LIN {X 0,Y 249.052,Z 167.452,A -85,B 0,C 180,E1 -18878.627,E2 -18878.627} C_VEL
LIN {X 0,Y 249.159,Z 167.445,A -85,B 0,C 180,E1 -18883.615,E2 -18883.615} C_VEL
LIN {X 0,Y 249.22,Z 167.437,A -85,B 0,C 180,E1 -18888.614,E2 -18888.614} C_VEL
LIN {X 0,Y 249.416,Z 167.401,A -85,B 0,C 180,E1 -18891.9,E2 -18891.9} C_VEL
LIN {X 0,Y 249.265,Z 167.429,A -85,B 0,C 180,E1 -18895.147,E2 -18895.147} C_VEL
LIN {X 0,Y 249.662,Z 167.381,A -85,B 0,C 180,E1 -18898.386,E2 -18898.386} C_VEL
LIN {X 0,Y 249.67,Z 167.37,A -85,B 0,C 180,E1 -18901.612,E2 -18901.612} C_VEL
LIN {X 0,Y 249.428,Z 167.402,A -85,B 0,C 180,E1 -18906.546,E2 -18906.546} C_VEL
LIN {X 0,Y 249.344,Z 167.415,A -85,B 0,C 180,E1 -18909.736,E2 -18909.736} C_VEL
LIN {X 0,Y 249.183,Z 167.435,A -85,B 0,C 180,E1 -18914.704,E2 -18914.704} C_VEL
LIN {X 0,Y 249.118,Z 167.445,A -85,B 0,C 180,E1 -18918.078,E2 -18918.078} C_VEL
LIN {X 0,Y 249.083,Z 167.452,A -85,B 0,C 180,E1 -18921.518,E2 -18921.518} C_VEL
LIN {X 0,Y 249.117,Z 167.45,A -85,B 0,C 180,E1 -18925.475,E2 -18925.475} C_VEL
LIN {X 0,Y 249.05,Z 167.46,A -85,B 0,C 180,E1 -18930.102,E2 -18930.102} C_VEL
LIN {X 0,Y 249.071,Z 167.695,A -85,B 0,C 180,E1 -18930.523,E2 -18930.523} C_VEL
LIN {X 0,Y 249.432,Z 169.077,A -85,B 0,C 180,E1 -18931.179,E2 -18931.179} C_VEL
LIN {X 0,Y 252.028,Z 173,A -85,B 0,C 180,E1 -18931.947,E2 -18931.947} C_VEL
LIN {X 0,Y 253.509,Z 175.144,A -85,B 0,C 180,E1 -18932.37,E2 -18932.37} C_VEL
LIN {X 0,Y 260.713,Z 186.536,A -85,B 0,C 180,E1 -18934.354,E2 -18934.354} C_VEL
LIN {X 0,Y 269.126,Z 201.959,A -85,B 0,C 180,E1 -18936.505,E2 -18936.505} C_VEL
LIN {X 0,Y 275.328,Z 215.39,A -85,B 0,C 180,E1 -18938.036,E2 -18938.036} C_VEL
LIN {X 0,Y 272.536,Z 275.676,A -85,B 0,C 180,E1 -18939.662,E2 -18939.662} C_VEL
LIN {X 0,Y 271.152,Z 289.633,A -85,B 0,C 180,E1 -18940.333,E2 -18940.333} C_VEL
LIN {X 0,Y 269.51,Z 302.431,A -85,B 0,C 180,E1 -18941.293,E2 -18941.293} C_VEL
LIN {X 0,Y 267.486,Z 313.271,A -85,B 0,C 180,E1 -18942.357,E2 -18942.357} C_VEL
LIN {X 0,Y 265.177,Z 324.055,A -85,B 0,C 180,E1 -18943.733,E2 -18943.733} C_VEL
LIN {X 0,Y 262.562,Z 334.24,A -85,B 0,C 180,E1 -18945.361,E2 -18945.361} C_VEL
LIN {X 0,Y 259.944,Z 343.294,A -85,B 0,C 180,E1 -18947.168,E2 -18947.168} C_VEL
LIN {X 0,Y 257.103,Z 352.123,A -85,B 0,C 180,E1 -18949.396,E2 -18949.396} C_VEL
LIN {X 0,Y 254.695,Z 359.121,A -85,B 0,C 180,E1 -18951.621,E2 -18951.621} C_VEL
LIN {X 0,Y 252.375,Z 365.518,A -85,B 0,C 180,E1 -18954.211,E2 -18954.211} C_VEL
LIN {X 0,Y 250.551,Z 370.339,A -85,B 0,C 180,E1 -18956.782,E2 -18956.782} C_VEL
LIN {X 0,Y 249.074,Z 374.017,A -85,B 0,C 180,E1 -18959.476,E2 -18959.476} C_VEL
LIN {X 0,Y 248.275,Z 375.843,A -85,B 0,C 180,E1 -18961.344,E2 -18961.344} C_VEL
LIN {X 0,Y 247.697,Z 377.032,A -85,B 0,C 180,E1 -18963.001,E2 -18963.001} C_VEL
LIN {X 0,Y 247.134,Z 377.998,A -85,B 0,C 180,E1 -18965.505,E2 -18965.505} C_VEL
LIN {X 0,Y 246.776,Z 378.012,A -85,B 0,C 180,E1 -18968.27,E2 -18968.27} C_VEL
LIN {X 0,Y 246.746,Z 377.407,A -85,B 0,C 180,E1 -18970.037,E2 -18970.037} C_VEL
LIN {X 0,Y 246.719,Z 376.398,A -85,B 0,C 180,E1 -18971.739,E2 -18971.739} C_VEL
LIN {X 0,Y 246.848,Z 374.953,A -85,B 0,C 180,E1 -18973.459,E2 -18973.459} C_VEL
LIN {X 0,Y 247.272,Z 371.847,A -85,B 0,C 180,E1 -18976.048,E2 -18976.048} C_VEL
LIN {X 0,Y 247.792,Z 367.733,A -85,B 0,C 180,E1 -18978.549,E2 -18978.549} C_VEL
LIN {X 0,Y 248.725,Z 361.306,A -85,B 0,C 180,E1 -18981.473,E2 -18981.473} C_VEL
LIN {X 0,Y 249.811,Z 354.327,A -85,B 0,C 180,E1 -18983.944,E2 -18983.944} C_VEL
LIN {X 0,Y 250.983,Z 347.179,A -85,B 0,C 180,E1 -18985.986,E2 -18985.986} C_VEL
LIN {X 0,Y 252.381,Z 338.546,A -85,B 0,C 180,E1 -18988.005,E2 -18988.005} C_VEL
LIN {X 0,Y 254.085,Z 327.819,A -85,B 0,C 180,E1 -18990,E2 -18990} C_VEL
LIN {X 0,Y 255.511,Z 317.218,A -85,B 0,C 180,E1 -18991.576,E2 -18991.576} C_VEL
LIN {X 0,Y 256.936,Z 305.486,A -85,B 0,C 180,E1 -18992.94,E2 -18992.94} C_VEL
LIN {X 0,Y 258.068,Z 293.324,A -85,B 0,C 180,E1 -18994.002,E2 -18994.002} C_VEL
LIN {X 0,Y 258.95,Z 280.161,A -85,B 0,C 180,E1 -18994.817,E2 -18994.817} C_VEL
LIN {X 0,Y 259.553,Z 267.449,A -85,B 0,C 180,E1 -18995.292,E2 -18995.292} C_VEL
LIN {X 0,Y 261.586,Z 201.975,A -85,B 0,C 180,E1 -18997.076,E2 -18997.076} C_VEL
LIN {X 0,Y 259.605,Z 195.135,A -85,B 0,C 180,E1 -18997.457,E2 -18997.457} C_VEL
LIN {X 0,Y 251.738,Z 173.167,A -85,B 0,C 180,E1 -18998.873,E2 -18998.873} C_VEL
LIN {X 0,Y 249.492,Z 168.039,A -85,B 0,C 180,E1 -18999.256,E2 -18999.256} C_VEL
LIN {X 0,Y 249.385,Z 167.421,A -85,B 0,C 180,E1 -18999.296,E2 -18999.296} C_VEL
LIN {X 0,Y 249.138,Z 167.452,A -85,B 0,C 180,E1 -19004.708,E2 -19004.708} C_VEL
LIN {X 0,Y 249.072,Z 167.46,A -85,B 0,C 180,E1 -19008.083,E2 -19008.083} C_VEL
LIN {X 0,Y 249.038,Z 167.46,A -85,B 0,C 180,E1 -19011.523,E2 -19011.523} C_VEL
LIN {X 0,Y 249.035,Z 167.435,A -85,B 0,C 180,E1 -19015.438,E2 -19015.438} C_VEL
LIN {X 0,Y 249.021,Z 167.457,A -85,B 0,C 180,E1 -19018.969,E2 -19018.969} C_VEL
LIN {X 0,Y 249.023,Z 167.464,A -85,B 0,C 180,E1 -19022.428,E2 -19022.428} C_VEL
LIN {X 0,Y 249.024,Z 167.451,A -85,B 0,C 180,E1 -19026.347,E2 -19026.347} C_VEL
LIN {X 0,Y 248.977,Z 167.47,A -85,B 0,C 180,E1 -19030.485,E2 -19030.485} C_VEL
LIN {X 0,Y 248.96,Z 167.462,A -85,B 0,C 180,E1 -19034.89,E2 -19034.89} C_VEL
LIN {X 0,Y 248.978,Z 167.455,A -85,B 0,C 180,E1 -19037.356,E2 -19037.356} C_VEL
LIN {X 0,Y 249.04,Z 167.461,A -85,B 0,C 180,E1 -19042.202,E2 -19042.202} C_VEL
LIN {X 0,Y 249.043,Z 167.457,A -85,B 0,C 180,E1 -19045.64,E2 -19045.64} C_VEL
LIN {X 0,Y 248.994,Z 167.445,A -85,B 0,C 180,E1 -19049.466,E2 -19049.466} C_VEL
LIN {X 0,Y 249.014,Z 167.455,A -85,B 0,C 180,E1 -19053.156,E2 -19053.156} C_VEL
LIN {X 0,Y 249.006,Z 167.467,A -85,B 0,C 180,E1 -19056.726,E2 -19056.726} C_VEL
LIN {X 0,Y 249.042,Z 167.463,A -85,B 0,C 180,E1 -19060.207,E2 -19060.207} C_VEL
LIN {X 0,Y 249.16,Z 167.442,A -85,B 0,C 180,E1 -19063.617,E2 -19063.617} C_VEL
LIN {X 0,Y 249.218,Z 167.439,A -85,B 0,C 180,E1 -19068.616,E2 -19068.616} C_VEL
LIN {X 0,Y 249.418,Z 167.41,A -85,B 0,C 180,E1 -19071.902,E2 -19071.902} C_VEL
LIN {X 0,Y 249.259,Z 167.435,A -85,B 0,C 180,E1 -19075.149,E2 -19075.149} C_VEL
LIN {X 0,Y 249.658,Z 167.381,A -85,B 0,C 180,E1 -19078.388,E2 -19078.388} C_VEL
LIN {X 0,Y 249.66,Z 167.384,A -85,B 0,C 180,E1 -19081.614,E2 -19081.614} C_VEL
LIN {X 0,Y 249.429,Z 167.411,A -85,B 0,C 180,E1 -19086.472,E2 -19086.472} C_VEL
LIN {X 0,Y 249.402,Z 167.412,A -85,B 0,C 180,E1 -19088.405,E2 -19088.405} C_VEL
LIN {X 0,Y 248.673,Z 167.508,A -85,B 0,C 180,E1 -19089.751,E2 -19089.751} C_VEL
LIN {X 0,Y 245.735,Z 167.876,A -85,B 0,C 180,E1 -19091.942,E2 -19091.942} C_VEL
LIN {X 0,Y 243.258,Z 168.185,A -85,B 0,C 180,E1 -19093.726,E2 -19093.726} C_VEL
LIN {X 0,Y 242.186,Z 168.315,A -85,B 0,C 180,E1 -19095.112,E2 -19095.112} C_VEL
LIN {X 0,Y 242.093,Z 168.323,A -85,B 0,C 180,E1 -19095.583,E2 -19095.583} C_VEL
LIN {X 0,Y 241.989,Z 168.34,A -85,B 0,C 180,E1 -19100.397,E2 -19100.397} C_VEL
LIN {X 0,Y 242.028,Z 168.335,A -85,B 0,C 180,E1 -19103.988,E2 -19103.988} C_VEL
LIN {X 0,Y 241.972,Z 168.342,A -85,B 0,C 180,E1 -19107.693,E2 -19107.693} C_VEL
LIN {X 0,Y 241.957,Z 168.345,A -85,B 0,C 180,E1 -19111.524,E2 -19111.524} C_VEL
LIN {X 0,Y 241.982,Z 168.342,A -85,B 0,C 180,E1 -19115.588,E2 -19115.588} C_VEL
LIN {X 0,Y 241.944,Z 168.348,A -85,B 0,C 180,E1 -19119.723,E2 -19119.723} C_VEL
LIN {X 0,Y 241.901,Z 168.355,A -85,B 0,C 180,E1 -19124.21,E2 -19124.21} C_VEL
LIN {X 0,Y 241.922,Z 168.351,A -85,B 0,C 180,E1 -19128.074,E2 -19128.074} C_VEL
LIN {X 0,Y 241.99,Z 168.339,A -85,B 0,C 180,E1 -19132.417,E2 -19132.417} C_VEL
LIN {X 0,Y 242.046,Z 168.546,A -85,B 0,C 180,E1 -19134.754,E2 -19134.754} C_VEL
LIN {X 0,Y 244.315,Z 179.21,A -85,B 0,C 180,E1 -19138.815,E2 -19138.815} C_VEL
LIN {X 0,Y 245.111,Z 183.189,A -85,B 0,C 180,E1 -19140.272,E2 -19140.272} C_VEL
LIN {X 0,Y 249.449,Z 195.846,A -85,B 0,C 180,E1 -19141.11,E2 -19141.11} C_VEL
LIN {X 0,Y 254.127,Z 234.244,A -85,B 0,C 180,E1 -19142.738,E2 -19142.738} C_VEL
LIN {X 0,Y 252.285,Z 292.507,A -85,B 0,C 180,E1 -19144.418,E2 -19144.418} C_VEL
LIN {X 0,Y 251.321,Z 306.261,A -85,B 0,C 180,E1 -19145.144,E2 -19145.144} C_VEL
LIN {X 0,Y 249.948,Z 319.146,A -85,B 0,C 180,E1 -19146.159,E2 -19146.159} C_VEL
LIN {X 0,Y 248.279,Z 331.738,A -85,B 0,C 180,E1 -19147.533,E2 -19147.533} C_VEL
LIN {X 0,Y 246.562,Z 342.976,A -85,B 0,C 180,E1 -19149.126,E2 -19149.126} C_VEL
LIN {X 0,Y 245.004,Z 353.19,A -85,B 0,C 180,E1 -19150.978,E2 -19150.978} C_VEL
LIN {X 0,Y 243.858,Z 360.177,A -85,B 0,C 180,E1 -19152.501,E2 -19152.501} C_VEL
LIN {X 0,Y 242.455,Z 369.09,A -85,B 0,C 180,E1 -19154.877,E2 -19154.877} C_VEL
LIN {X 0,Y 241.179,Z 376.588,A -85,B 0,C 180,E1 -19157.376,E2 -19157.376} C_VEL
LIN {X 0,Y 240.48,Z 382.608,A -85,B 0,C 180,E1 -19159.901,E2 -19159.901} C_VEL
LIN {X 0,Y 240.04,Z 387.334,A -85,B 0,C 180,E1 -19162.429,E2 -19162.429} C_VEL
LIN {X 0,Y 239.846,Z 391.044,A -85,B 0,C 180,E1 -19165.059,E2 -19165.059} C_VEL
LIN {X 0,Y 239.88,Z 392.734,A -85,B 0,C 180,E1 -19166.64,E2 -19166.64} C_VEL
LIN {X 0,Y 239.951,Z 394.089,A -85,B 0,C 180,E1 -19168.321,E2 -19168.321} C_VEL
LIN {X 0,Y 239.959,Z 395.035,A -85,B 0,C 180,E1 -19170,E2 -19170} C_VEL
LIN {X 0,Y 239.925,Z 395.584,A -85,B 0,C 180,E1 -19171.678,E2 -19171.678} C_VEL
LIN {X 0,Y 239.804,Z 395.501,A -85,B 0,C 180,E1 -19174.823,E2 -19174.823} C_VEL
LIN {X 0,Y 239.904,Z 394.768,A -85,B 0,C 180,E1 -19176.729,E2 -19176.729} C_VEL
LIN {X 0,Y 240.627,Z 392.277,A -85,B 0,C 180,E1 -19180.093,E2 -19180.093} C_VEL
LIN {X 0,Y 241.547,Z 389.295,A -85,B 0,C 180,E1 -19182.604,E2 -19182.604} C_VEL
LIN {X 0,Y 242.961,Z 385.297,A -85,B 0,C 180,E1 -19185.09,E2 -19185.09} C_VEL
LIN {X 0,Y 245.269,Z 379.2,A -85,B 0,C 180,E1 -19187.941,E2 -19187.941} C_VEL
LIN {X 0,Y 247.576,Z 372.206,A -85,B 0,C 180,E1 -19190.481,E2 -19190.481} C_VEL
LIN {X 0,Y 250.288,Z 364.407,A -85,B 0,C 180,E1 -19192.712,E2 -19192.712} C_VEL
LIN {X 0,Y 253.066,Z 356.079,A -85,B 0,C 180,E1 -19194.618,E2 -19194.618} C_VEL
LIN {X 0,Y 256.057,Z 345.877,A -85,B 0,C 180,E1 -19196.488,E2 -19196.488} C_VEL
LIN {X 0,Y 258.721,Z 335.819,A -85,B 0,C 180,E1 -19197.942,E2 -19197.942} C_VEL
LIN {X 0,Y 261.255,Z 324.883,A -85,B 0,C 180,E1 -19199.181,E2 -19199.181} C_VEL
LIN {X 0,Y 263.592,Z 312.804,A -85,B 0,C 180,E1 -19200.215,E2 -19200.215} C_VEL
LIN {X 0,Y 265.434,Z 300.26,A -85,B 0,C 180,E1 -19200.974,E2 -19200.974} C_VEL
LIN {X 0,Y 266.549,Z 287.421,A -85,B 0,C 180,E1 -19201.493,E2 -19201.493} C_VEL
LIN {X 0,Y 268.646,Z 237.587,A -85,B 0,C 180,E1 -19202.879,E2 -19202.879} C_VEL
LIN {X 0,Y 265.876,Z 220.013,A -85,B 0,C 180,E1 -19203.988,E2 -19203.988} C_VEL
LIN {X 0,Y 260.082,Z 207.142,A -85,B 0,C 180,E1 -19205.547,E2 -19205.547} C_VEL
LIN {X 0,Y 253.89,Z 195.175,A -85,B 0,C 180,E1 -19207.291,E2 -19207.291} C_VEL
LIN {X 0,Y 250.768,Z 189.794,A -85,B 0,C 180,E1 -19208.201,E2 -19208.201} C_VEL
LIN {X 0,Y 248.439,Z 185.77,A -85,B 0,C 180,E1 -19208.904,E2 -19208.904} C_VEL
LIN {X 0,Y 245.726,Z 181.065,A -85,B 0,C 180,E1 -19209.766,E2 -19209.766} C_VEL
LIN {X 0,Y 243.463,Z 173.399,A -85,B 0,C 180,E1 -19213.852,E2 -19213.852} C_VEL
LIN {X 0,Y 241.943,Z 168.344,A -85,B 0,C 180,E1 -19216.923,E2 -19216.923} C_VEL
LIN {X 0,Y 241.991,Z 168.336,A -85,B 0,C 180,E1 -19221.642,E2 -19221.642} C_VEL
LIN {X 0,Y 241.987,Z 168.338,A -85,B 0,C 180,E1 -19224.488,E2 -19224.488} C_VEL
LIN {X 0,Y 241.954,Z 168.337,A -85,B 0,C 180,E1 -19228.476,E2 -19228.476} C_VEL
LIN {X 0,Y 241.959,Z 168.335,A -85,B 0,C 180,E1 -19232.306,E2 -19232.306} C_VEL
LIN {X 0,Y 241.984,Z 168.336,A -85,B 0,C 180,E1 -19236.007,E2 -19236.007} C_VEL
LIN {X 0,Y 241.984,Z 168.341,A -85,B 0,C 180,E1 -19239.602,E2 -19239.602} C_VEL
LIN {X 0,Y 242.107,Z 168.319,A -85,B 0,C 180,E1 -19243.324,E2 -19243.324} C_VEL
LIN {X 0,Y 242.154,Z 168.312,A -85,B 0,C 180,E1 -19248.277,E2 -19248.277} C_VEL
LIN {X 0,Y 242.37,Z 168.278,A -85,B 0,C 180,E1 -19251.663,E2 -19251.663} C_VEL
LIN {X 0,Y 242.398,Z 168.284,A -85,B 0,C 180,E1 -19253.339,E2 -19253.339} C_VEL
LIN {X 0,Y 242.621,Z 168.257,A -85,B 0,C 180,E1 -19258.339,E2 -19258.339} C_VEL
LIN {X 0,Y 242.631,Z 168.246,A -85,B 0,C 180,E1 -19261.659,E2 -19261.659} C_VEL
LIN {X 0,Y 242.404,Z 168.278,A -85,B 0,C 180,E1 -19266.659,E2 -19266.659} C_VEL
LIN {X 0,Y 242.268,Z 168.295,A -85,B 0,C 180,E1 -19270.023,E2 -19270.023} C_VEL
LIN {X 0,Y 242.139,Z 168.313,A -85,B 0,C 180,E1 -19275.142,E2 -19275.142} C_VEL
LIN {X 0,Y 242.057,Z 168.324,A -85,B 0,C 180,E1 -19278.624,E2 -19278.624} C_VEL
LIN {X 0,Y 242.006,Z 168.333,A -85,B 0,C 180,E1 -19282.18,E2 -19282.18} C_VEL
LIN {X 0,Y 242.066,Z 168.33,A -85,B 0,C 180,E1 -19285.837,E2 -19285.837} C_VEL
LIN {X 0,Y 242.062,Z 168.433,A -85,B 0,C 180,E1 -19288.936,E2 -19288.936} C_VEL
LIN {X 0,Y 242.287,Z 169.476,A -85,B 0,C 180,E1 -19289.422,E2 -19289.422} C_VEL
LIN {X 0,Y 243.54,Z 171.918,A -85,B 0,C 180,E1 -19289.853,E2 -19289.853} C_VEL
LIN {X 0,Y 245.704,Z 174.554,A -85,B 0,C 180,E1 -19290.51,E2 -19290.51} C_VEL
LIN {X 0,Y 250.027,Z 180.984,A -85,B 0,C 180,E1 -19291.815,E2 -19291.815} C_VEL
LIN {X 0,Y 255.207,Z 189.289,A -85,B 0,C 180,E1 -19293.308,E2 -19293.308} C_VEL
LIN {X 0,Y 261.074,Z 199.751,A -85,B 0,C 180,E1 -19294.922,E2 -19294.922} C_VEL
LIN {X 0,Y 267.14,Z 211.817,A -85,B 0,C 180,E1 -19296.498,E2 -19296.498} C_VEL
LIN {X 0,Y 269.609,Z 217.281,A -85,B 0,C 180,E1 -19297.129,E2 -19297.129} C_VEL
LIN {X 0,Y 266.947,Z 275.288,A -85,B 0,C 180,E1 -19298.732,E2 -19298.732} C_VEL
LIN {X 0,Y 265.549,Z 288.86,A -85,B 0,C 180,E1 -19299.371,E2 -19299.371} C_VEL
LIN {X 0,Y 263.88,Z 301.755,A -85,B 0,C 180,E1 -19300.326,E2 -19300.326} C_VEL
LIN {X 0,Y 261.617,Z 313.504,A -85,B 0,C 180,E1 -19301.484,E2 -19301.484} C_VEL
LIN {X 0,Y 259.133,Z 324.573,A -85,B 0,C 180,E1 -19302.923,E2 -19302.923} C_VEL
LIN {X 0,Y 256.454,Z 334.59,A -85,B 0,C 180,E1 -19304.56,E2 -19304.56} C_VEL
LIN {X 0,Y 253.353,Z 344.637,A -85,B 0,C 180,E1 -19306.641,E2 -19306.641} C_VEL
LIN {X 0,Y 250.602,Z 352.719,A -85,B 0,C 180,E1 -19308.762,E2 -19308.762} C_VEL
LIN {X 0,Y 247.74,Z 360.588,A -85,B 0,C 180,E1 -19311.383,E2 -19311.383} C_VEL
LIN {X 0,Y 245.347,Z 366.676,A -85,B 0,C 180,E1 -19314.04,E2 -19314.04} C_VEL
LIN {X 0,Y 243.369,Z 371.544,A -85,B 0,C 180,E1 -19316.871,E2 -19316.871} C_VEL
LIN {X 0,Y 242.417,Z 373.766,A -85,B 0,C 180,E1 -19318.544,E2 -19318.544} C_VEL
LIN {X 0,Y 241.339,Z 376.076,A -85,B 0,C 180,E1 -19320.881,E2 -19320.881} C_VEL
LIN {X 0,Y 240.342,Z 377.928,A -85,B 0,C 180,E1 -19323.984,E2 -19323.984} C_VEL
LIN {X 0,Y 239.986,Z 378.348,A -85,B 0,C 180,E1 -19325.796,E2 -19325.796} C_VEL
LIN {X 0,Y 239.743,Z 378.327,A -85,B 0,C 180,E1 -19327.599,E2 -19327.599} C_VEL
LIN {X 0,Y 239.66,Z 377.713,A -85,B 0,C 180,E1 -19329.781,E2 -19329.781} C_VEL
LIN {X 0,Y 239.691,Z 375.603,A -85,B 0,C 180,E1 -19332.95,E2 -19332.95} C_VEL
LIN {X 0,Y 239.981,Z 373.331,A -85,B 0,C 180,E1 -19335.107,E2 -19335.107} C_VEL
LIN {X 0,Y 240.429,Z 370.208,A -85,B 0,C 180,E1 -19337.336,E2 -19337.336} C_VEL
LIN {X 0,Y 241.199,Z 364.437,A -85,B 0,C 180,E1 -19340.398,E2 -19340.398} C_VEL
LIN {X 0,Y 242.18,Z 358.266,A -85,B 0,C 180,E1 -19342.916,E2 -19342.916} C_VEL
LIN {X 0,Y 243.433,Z 350.48,A -85,B 0,C 180,E1 -19345.447,E2 -19345.447} C_VEL
LIN {X 0,Y 244.838,Z 342.453,A -85,B 0,C 180,E1 -19347.533,E2 -19347.533} C_VEL
LIN {X 0,Y 246.471,Z 333.018,A -85,B 0,C 180,E1 -19349.516,E2 -19349.516} C_VEL
LIN {X 0,Y 248.128,Z 321.729,A -85,B 0,C 180,E1 -19351.42,E2 -19351.42} C_VEL
LIN {X 0,Y 249.613,Z 311.095,A -85,B 0,C 180,E1 -19352.825,E2 -19352.825} C_VEL
LIN {X 0,Y 250.914,Z 298.386,A -85,B 0,C 180,E1 -19354.116,E2 -19354.116} C_VEL
LIN {X 0,Y 251.907,Z 285.726,A -85,B 0,C 180,E1 -19355.052,E2 -19355.052} C_VEL
LIN {X 0,Y 252.66,Z 273.673,A -85,B 0,C 180,E1 -19355.637,E2 -19355.637} C_VEL
LIN {X 0,Y 254.94,Z 202.652,A -85,B 0,C 180,E1 -19357.649,E2 -19357.649} C_VEL
LIN {X 0,Y 246.322,Z 177.811,A -85,B 0,C 180,E1 -19359.264,E2 -19359.264} C_VEL
LIN {X 0,Y 242.429,Z 169.195,A -85,B 0,C 180,E1 -19359.946,E2 -19359.946} C_VEL
LIN {X 0,Y 242.255,Z 168.309,A -85,B 0,C 180,E1 -19360.025,E2 -19360.025} C_VEL
LIN {X 0,Y 242.098,Z 168.33,A -85,B 0,C 180,E1 -19365.146,E2 -19365.146} C_VEL
LIN {X 0,Y 242.01,Z 168.338,A -85,B 0,C 180,E1 -19368.63,E2 -19368.63} C_VEL
LIN {X 0,Y 241.968,Z 168.336,A -85,B 0,C 180,E1 -19372.185,E2 -19372.185} C_VEL
LIN {X 0,Y 241.982,Z 168.312,A -85,B 0,C 180,E1 -19375.827,E2 -19375.827} C_VEL
LIN {X 0,Y 241.96,Z 168.341,A -85,B 0,C 180,E1 -19379.59,E2 -19379.59} C_VEL
LIN {X 0,Y 241.976,Z 168.341,A -85,B 0,C 180,E1 -19383.494,E2 -19383.494} C_VEL
LIN {X 0,Y 241.981,Z 168.336,A -85,B 0,C 180,E1 -19387.584,E2 -19387.584} C_VEL
LIN {X 0,Y 241.906,Z 168.35,A -85,B 0,C 180,E1 -19391.93,E2 -19391.93} C_VEL
LIN {X 0,Y 241.899,Z 168.333,A -85,B 0,C 180,E1 -19396.581,E2 -19396.581} C_VEL
LIN {X 0,Y 241.992,Z 168.338,A -85,B 0,C 180,E1 -19401.642,E2 -19401.642} C_VEL
LIN {X 0,Y 241.979,Z 168.343,A -85,B 0,C 180,E1 -19404.489,E2 -19404.489} C_VEL
LIN {X 0,Y 241.948,Z 168.327,A -85,B 0,C 180,E1 -19408.477,E2 -19408.477} C_VEL
LIN {X 0,Y 241.951,Z 168.325,A -85,B 0,C 180,E1 -19412.307,E2 -19412.307} C_VEL
LIN {X 0,Y 241.957,Z 168.341,A -85,B 0,C 180,E1 -19416.006,E2 -19416.006} C_VEL
LIN {X 0,Y 241.983,Z 168.341,A -85,B 0,C 180,E1 -19419.604,E2 -19419.604} C_VEL
LIN {X 0,Y 242.107,Z 168.32,A -85,B 0,C 180,E1 -19423.326,E2 -19423.326} C_VEL
LIN {X 0,Y 242.151,Z 168.321,A -85,B 0,C 180,E1 -19428.279,E2 -19428.279} C_VEL
LIN {X 0,Y 242.371,Z 168.286,A -85,B 0,C 180,E1 -19431.665,E2 -19431.665} C_VEL
LIN {X 0,Y 242.4,Z 168.287,A -85,B 0,C 180,E1 -19433.341,E2 -19433.341} C_VEL
LIN {X 0,Y 242.618,Z 168.258,A -85,B 0,C 180,E1 -19438.341,E2 -19438.341} C_VEL
LIN {X 0,Y 242.62,Z 168.261,A -85,B 0,C 180,E1 -19441.661,E2 -19441.661} C_VEL
LIN {X 0,Y 242.4,Z 168.286,A -85,B 0,C 180,E1 -19446.661,E2 -19446.661} C_VEL
LIN {X 0,Y 242.27,Z 168.306,A -85,B 0,C 180,E1 -19450.024,E2 -19450.024} C_VEL
LIN {X 0,Y 242.111,Z 168.324,A -85,B 0,C 180,E1 -19455.145,E2 -19455.145} C_VEL
LIN {X 0,Y 242.093,Z 168.323,A -85,B 0,C 180,E1 -19455.583,E2 -19455.583} C_VEL
LIN {X 0,Y 241.41,Z 168.409,A -85,B 0,C 180,E1 -19456.969,E2 -19456.969} C_VEL
LIN {X 0,Y 238.554,Z 168.77,A -85,B 0,C 180,E1 -19459.231,E2 -19459.231} C_VEL
LIN {X 0,Y 236.115,Z 169.079,A -85,B 0,C 180,E1 -19461.073,E2 -19461.073} C_VEL
LIN {X 0,Y 235.04,Z 169.209,A -85,B 0,C 180,E1 -19462.502,E2 -19462.502} C_VEL
LIN {X 0,Y 234.936,Z 169.219,A -85,B 0,C 180,E1 -19462.987,E2 -19462.987} C_VEL
LIN {X 0,Y 234.949,Z 169.218,A -85,B 0,C 180,E1 -19466.661,E2 -19466.661} C_VEL
LIN {X 0,Y 234.903,Z 169.224,A -85,B 0,C 180,E1 -19470.573,E2 -19470.573} C_VEL
LIN {X 0,Y 234.93,Z 169.222,A -85,B 0,C 180,E1 -19474.639,E2 -19474.639} C_VEL
LIN {X 0,Y 234.916,Z 169.226,A -85,B 0,C 180,E1 -19478.935,E2 -19478.935} C_VEL
LIN {X 0,Y 234.858,Z 169.232,A -85,B 0,C 180,E1 -19483.494,E2 -19483.494} C_VEL
LIN {X 0,Y 234.865,Z 169.233,A -85,B 0,C 180,E1 -19486.508,E2 -19486.508} C_VEL
LIN {X 0,Y 234.922,Z 169.222,A -85,B 0,C 180,E1 -19491.079,E2 -19491.079} C_VEL
LIN {X 0,Y 234.959,Z 169.302,A -85,B 0,C 180,E1 -19494.185,E2 -19494.185} C_VEL
LIN {X 0,Y 237.115,Z 179.284,A -85,B 0,C 180,E1 -19498.13,E2 -19498.13} C_VEL
LIN {X 0,Y 237.915,Z 183.179,A -85,B 0,C 180,E1 -19499.521,E2 -19499.521} C_VEL
LIN {X 0,Y 243.059,Z 197.717,A -85,B 0,C 180,E1 -19500.533,E2 -19500.533} C_VEL
LIN {X 0,Y 247.492,Z 233.694,A -85,B 0,C 180,E1 -19502.121,E2 -19502.121} C_VEL
LIN {X 0,Y 245.638,Z 291.986,A -85,B 0,C 180,E1 -19503.845,E2 -19503.845} C_VEL
LIN {X 0,Y 244.706,Z 305.061,A -85,B 0,C 180,E1 -19504.538,E2 -19504.538} C_VEL
LIN {X 0,Y 243.439,Z 317.159,A -85,B 0,C 180,E1 -19505.48,E2 -19505.48} C_VEL
LIN {X 0,Y 241.957,Z 328.598,A -85,B 0,C 180,E1 -19506.686,E2 -19506.686} C_VEL
LIN {X 0,Y 240.402,Z 339.073,A -85,B 0,C 180,E1 -19508.115,E2 -19508.115} C_VEL
LIN {X 0,Y 238.729,Z 348.786,A -85,B 0,C 180,E1 -19509.762,E2 -19509.762} C_VEL
LIN {X 0,Y 237.327,Z 357.082,A -85,B 0,C 180,E1 -19511.484,E2 -19511.484} C_VEL
LIN {X 0,Y 235.993,Z 365.313,A -85,B 0,C 180,E1 -19513.565,E2 -19513.565} C_VEL
LIN {X 0,Y 234.626,Z 373.53,A -85,B 0,C 180,E1 -19516.135,E2 -19516.135} C_VEL
LIN {X 0,Y 233.67,Z 380.122,A -85,B 0,C 180,E1 -19518.726,E2 -19518.726} C_VEL
LIN {X 0,Y 233.111,Z 385.34,A -85,B 0,C 180,E1 -19521.33,E2 -19521.33} C_VEL
LIN {X 0,Y 232.829,Z 389.364,A -85,B 0,C 180,E1 -19523.935,E2 -19523.935} C_VEL
LIN {X 0,Y 232.781,Z 392.316,A -85,B 0,C 180,E1 -19526.538,E2 -19526.538} C_VEL
LIN {X 0,Y 232.858,Z 393.716,A -85,B 0,C 180,E1 -19528.27,E2 -19528.27} C_VEL
LIN {X 0,Y 232.889,Z 394.695,A -85,B 0,C 180,E1 -19530,E2 -19530} C_VEL
LIN {X 0,Y 232.83,Z 395.275,A -85,B 0,C 180,E1 -19531.729,E2 -19531.729} C_VEL
LIN {X 0,Y 232.725,Z 395.322,A -85,B 0,C 180,E1 -19534.745,E2 -19534.745} C_VEL
LIN {X 0,Y 232.826,Z 394.585,A -85,B 0,C 180,E1 -19536.935,E2 -19536.935} C_VEL
LIN {X 0,Y 233.603,Z 392.171,A -85,B 0,C 180,E1 -19540.399,E2 -19540.399} C_VEL
LIN {X 0,Y 234.589,Z 389.245,A -85,B 0,C 180,E1 -19542.984,E2 -19542.984} C_VEL
LIN {X 0,Y 236.087,Z 385.328,A -85,B 0,C 180,E1 -19545.54,E2 -19545.54} C_VEL
LIN {X 0,Y 238.162,Z 380.311,A -85,B 0,C 180,E1 -19548.05,E2 -19548.05} C_VEL
LIN {X 0,Y 240.791,Z 372.902,A -85,B 0,C 180,E1 -19550.933,E2 -19550.933} C_VEL
LIN {X 0,Y 243.782,Z 364.795,A -85,B 0,C 180,E1 -19553.353,E2 -19553.353} C_VEL
LIN {X 0,Y 246.667,Z 356.594,A -85,B 0,C 180,E1 -19555.301,E2 -19555.301} C_VEL
LIN {X 0,Y 249.758,Z 346.629,A -85,B 0,C 180,E1 -19557.21,E2 -19557.21} C_VEL
LIN {X 0,Y 252.905,Z 335.38,A -85,B 0,C 180,E1 -19558.871,E2 -19558.871} C_VEL
LIN {X 0,Y 255.543,Z 324.402,A -85,B 0,C 180,E1 -19560.127,E2 -19560.127} C_VEL
LIN {X 0,Y 257.973,Z 312.258,A -85,B 0,C 180,E1 -19561.173,E2 -19561.173} C_VEL
LIN {X 0,Y 259.857,Z 299.561,A -85,B 0,C 180,E1 -19561.943,E2 -19561.943} C_VEL
LIN {X 0,Y 261.013,Z 286.461,A -85,B 0,C 180,E1 -19562.468,E2 -19562.468} C_VEL
LIN {X 0,Y 263.103,Z 238.663,A -85,B 0,C 180,E1 -19563.82,E2 -19563.82} C_VEL
LIN {X 0,Y 260.698,Z 223.005,A -85,B 0,C 180,E1 -19564.838,E2 -19564.838} C_VEL
LIN {X 0,Y 254.37,Z 208.912,A -85,B 0,C 180,E1 -19566.645,E2 -19566.645} C_VEL
LIN {X 0,Y 247.635,Z 196.106,A -85,B 0,C 180,E1 -19568.661,E2 -19568.661} C_VEL
LIN {X 0,Y 243.64,Z 189.504,A -85,B 0,C 180,E1 -19569.903,E2 -19569.903} C_VEL
LIN {X 0,Y 241.206,Z 185.458,A -85,B 0,C 180,E1 -19570.696,E2 -19570.696} C_VEL
LIN {X 0,Y 238.471,Z 180.958,A -85,B 0,C 180,E1 -19571.625,E2 -19571.625} C_VEL
LIN {X 0,Y 237.465,Z 177.609,A -85,B 0,C 180,E1 -19573.381,E2 -19573.381} C_VEL
LIN {X 0,Y 235.236,Z 170.655,A -85,B 0,C 180,E1 -19577.628,E2 -19577.628} C_VEL
LIN {X 0,Y 234.871,Z 169.225,A -85,B 0,C 180,E1 -19578.566,E2 -19578.566} C_VEL
LIN {X 0,Y 234.92,Z 169.221,A -85,B 0,C 180,E1 -19581.078,E2 -19581.078} C_VEL
LIN {X 0,Y 234.93,Z 169.211,A -85,B 0,C 180,E1 -19585.361,E2 -19585.361} C_VEL
LIN {X 0,Y 234.9,Z 169.213,A -85,B 0,C 180,E1 -19589.427,E2 -19589.427} C_VEL
LIN {X 0,Y 234.942,Z 169.207,A -85,B 0,C 180,E1 -19593.82,E2 -19593.82} C_VEL
LIN {X 0,Y 234.937,Z 169.214,A -85,B 0,C 180,E1 -19598.962,E2 -19598.962} C_VEL
LIN {X 0,Y 235.051,Z 169.195,A -85,B 0,C 180,E1 -19603.097,E2 -19603.097} C_VEL
LIN {X 0,Y 235.087,Z 169.189,A -85,B 0,C 180,E1 -19607.92,E2 -19607.92} C_VEL
LIN {X 0,Y 235.306,Z 169.159,A -85,B 0,C 180,E1 -19611.411,E2 -19611.411} C_VEL
LIN {X 0,Y 235.349,Z 169.159,A -85,B 0,C 180,E1 -19613.139,E2 -19613.139} C_VEL
LIN {X 0,Y 235.58,Z 169.133,A -85,B 0,C 180,E1 -19618.29,E2 -19618.29} C_VEL
LIN {X 0,Y 235.591,Z 169.123,A -85,B 0,C 180,E1 -19621.709,E2 -19621.709} C_VEL
LIN {X 0,Y 235.356,Z 169.157,A -85,B 0,C 180,E1 -19626.859,E2 -19626.859} C_VEL
LIN {X 0,Y 235.214,Z 169.172,A -85,B 0,C 180,E1 -19630.327,E2 -19630.327} C_VEL
LIN {X 0,Y 235.094,Z 169.194,A -85,B 0,C 180,E1 -19635.607,E2 -19635.607} C_VEL
LIN {X 0,Y 234.997,Z 169.206,A -85,B 0,C 180,E1 -19639.206,E2 -19639.206} C_VEL
LIN {X 0,Y 234.952,Z 169.215,A -85,B 0,C 180,E1 -19642.883,E2 -19642.883} C_VEL
LIN {X 0,Y 234.985,Z 169.36,A -85,B 0,C 180,E1 -19647.255,E2 -19647.255} C_VEL
LIN {X 0,Y 235.16,Z 170.206,A -85,B 0,C 180,E1 -19647.474,E2 -19647.474} C_VEL
LIN {X 0,Y 236.457,Z 172.755,A -85,B 0,C 180,E1 -19647.972,E2 -19647.972} C_VEL
LIN {X 0,Y 238.571,Z 174.895,A -85,B 0,C 180,E1 -19648.667,E2 -19648.667} C_VEL
LIN {X 0,Y 240.774,Z 178.262,A -85,B 0,C 180,E1 -19649.421,E2 -19649.421} C_VEL
LIN {X 0,Y 242.229,Z 180.277,A -85,B 0,C 180,E1 -19649.888,E2 -19649.888} C_VEL
LIN {X 0,Y 247.75,Z 188.516,A -85,B 0,C 180,E1 -19651.597,E2 -19651.597} C_VEL
LIN {X 0,Y 254.909,Z 200.88,A -85,B 0,C 180,E1 -19653.702,E2 -19653.702} C_VEL
LIN {X 0,Y 261.714,Z 214.342,A -85,B 0,C 180,E1 -19655.586,E2 -19655.586} C_VEL
LIN {X 0,Y 264.103,Z 219.738,A -85,B 0,C 180,E1 -19656.229,E2 -19656.229} C_VEL
LIN {X 0,Y 261.316,Z 276.128,A -85,B 0,C 180,E1 -19657.81,E2 -19657.81} C_VEL
LIN {X 0,Y 259.809,Z 290.022,A -85,B 0,C 180,E1 -19658.489,E2 -19658.489} C_VEL
LIN {X 0,Y 258.139,Z 302.204,A -85,B 0,C 180,E1 -19659.418,E2 -19659.418} C_VEL
LIN {X 0,Y 255.746,Z 314.064,A -85,B 0,C 180,E1 -19660.612,E2 -19660.612} C_VEL
LIN {X 0,Y 253.206,Z 324.949,A -85,B 0,C 180,E1 -19662.057,E2 -19662.057} C_VEL
LIN {X 0,Y 250.387,Z 334.936,A -85,B 0,C 180,E1 -19663.717,E2 -19663.717} C_VEL
LIN {X 0,Y 247.155,Z 344.965,A -85,B 0,C 180,E1 -19665.839,E2 -19665.839} C_VEL
LIN {X 0,Y 244.249,Z 353.065,A -85,B 0,C 180,E1 -19668.011,E2 -19668.011} C_VEL
LIN {X 0,Y 241.234,Z 360.891,A -85,B 0,C 180,E1 -19670.68,E2 -19670.68} C_VEL
LIN {X 0,Y 238.949,Z 366.402,A -85,B 0,C 180,E1 -19673.107,E2 -19673.107} C_VEL
LIN {X 0,Y 236.603,Z 371.771,A -85,B 0,C 180,E1 -19676.272,E2 -19676.272} C_VEL
LIN {X 0,Y 234.869,Z 375.49,A -85,B 0,C 180,E1 -19679.423,E2 -19679.423} C_VEL
LIN {X 0,Y 234.09,Z 376.974,A -85,B 0,C 180,E1 -19681.291,E2 -19681.291} C_VEL
LIN {X 0,Y 233.091,Z 378.496,A -85,B 0,C 180,E1 -19684.759,E2 -19684.759} C_VEL
LIN {X 0,Y 232.716,Z 378.644,A -85,B 0,C 180,E1 -19686.884,E2 -19686.884} C_VEL
LIN {X 0,Y 232.549,Z 378.01,A -85,B 0,C 180,E1 -19689.529,E2 -19689.529} C_VEL
LIN {X 0,Y 232.568,Z 376.252,A -85,B 0,C 180,E1 -19692.411,E2 -19692.411} C_VEL
LIN {X 0,Y 232.869,Z 373.752,A -85,B 0,C 180,E1 -19694.959,E2 -19694.959} C_VEL
LIN {X 0,Y 233.414,Z 369.738,A -85,B 0,C 180,E1 -19697.833,E2 -19697.833} C_VEL
LIN {X 0,Y 234.129,Z 364.783,A -85,B 0,C 180,E1 -19700.497,E2 -19700.497} C_VEL
LIN {X 0,Y 235.143,Z 358.52,A -85,B 0,C 180,E1 -19703.134,E2 -19703.134} C_VEL
LIN {X 0,Y 236.466,Z 350.726,A -85,B 0,C 180,E1 -19705.739,E2 -19705.739} C_VEL
LIN {X 0,Y 237.921,Z 342.695,A -85,B 0,C 180,E1 -19707.884,E2 -19707.884} C_VEL
LIN {X 0,Y 239.689,Z 332.848,A -85,B 0,C 180,E1 -19710,E2 -19710} C_VEL
LIN {X 0,Y 241.321,Z 321.966,A -85,B 0,C 180,E1 -19711.878,E2 -19711.878} C_VEL
LIN {X 0,Y 242.855,Z 311.326,A -85,B 0,C 180,E1 -19713.318,E2 -19713.318} C_VEL
LIN {X 0,Y 244.198,Z 298.615,A -85,B 0,C 180,E1 -19714.643,E2 -19714.643} C_VEL
LIN {X 0,Y 245.225,Z 285.951,A -85,B 0,C 180,E1 -19715.603,E2 -19715.603} C_VEL
LIN {X 0,Y 246.018,Z 273.854,A -85,B 0,C 180,E1 -19716.201,E2 -19716.201} C_VEL
LIN {X 0,Y 248.326,Z 203.809,A -85,B 0,C 180,E1 -19718.237,E2 -19718.237} C_VEL
LIN {X 0,Y 240.188,Z 180.533,A -85,B 0,C 180,E1 -19719.812,E2 -19719.812} C_VEL
LIN {X 0,Y 235.252,Z 169.807,A -85,B 0,C 180,E1 -19720.712,E2 -19720.712} C_VEL
LIN {X 0,Y 235.137,Z 169.196,A -85,B 0,C 180,E1 -19720.751,E2 -19720.751} C_VEL
LIN {X 0,Y 235.036,Z 169.21,A -85,B 0,C 180,E1 -19725.612,E2 -19725.612} C_VEL
LIN {X 0,Y 234.952,Z 169.218,A -85,B 0,C 180,E1 -19729.211,E2 -19729.211} C_VEL
LIN {X 0,Y 234.903,Z 169.209,A -85,B 0,C 180,E1 -19732.889,E2 -19732.889} C_VEL
LIN {X 0,Y 234.901,Z 169.198,A -85,B 0,C 180,E1 -19736.666,E2 -19736.666} C_VEL
LIN {X 0,Y 234.892,Z 169.223,A -85,B 0,C 180,E1 -19740.574,E2 -19740.574} C_VEL
LIN {X 0,Y 234.923,Z 169.217,A -85,B 0,C 180,E1 -19744.64,E2 -19744.64} C_VEL
LIN {X 0,Y 234.91,Z 169.22,A -85,B 0,C 180,E1 -19748.936,E2 -19748.936} C_VEL
LIN {X 0,Y 234.852,Z 169.224,A -85,B 0,C 180,E1 -19753.495,E2 -19753.495} C_VEL
LIN {X 0,Y 234.851,Z 169.21,A -85,B 0,C 180,E1 -19756.507,E2 -19756.507} C_VEL
LIN {X 0,Y 234.917,Z 169.221,A -85,B 0,C 180,E1 -19761.08,E2 -19761.08} C_VEL
LIN {X 0,Y 234.925,Z 169.215,A -85,B 0,C 180,E1 -19765.362,E2 -19765.362} C_VEL
LIN {X 0,Y 234.895,Z 169.198,A -85,B 0,C 180,E1 -19769.428,E2 -19769.428} C_VEL
LIN {X 0,Y 234.94,Z 169.206,A -85,B 0,C 180,E1 -19773.822,E2 -19773.822} C_VEL
LIN {X 0,Y 234.936,Z 169.219,A -85,B 0,C 180,E1 -19778.964,E2 -19778.964} C_VEL
LIN {X 0,Y 235.051,Z 169.198,A -85,B 0,C 180,E1 -19783.099,E2 -19783.099} C_VEL
LIN {X 0,Y 235.083,Z 169.203,A -85,B 0,C 180,E1 -19787.921,E2 -19787.921} C_VEL
LIN {X 0,Y 235.308,Z 169.165,A -85,B 0,C 180,E1 -19791.412,E2 -19791.412} C_VEL
LIN {X 0,Y 235.35,Z 169.165,A -85,B 0,C 180,E1 -19793.141,E2 -19793.141} C_VEL
LIN {X 0,Y 235.577,Z 169.135,A -85,B 0,C 180,E1 -19798.291,E2 -19798.291} C_VEL
LIN {X 0,Y 235.579,Z 169.138,A -85,B 0,C 180,E1 -19801.71,E2 -19801.71} C_VEL
LIN {X 0,Y 235.351,Z 169.164,A -85,B 0,C 180,E1 -19806.861,E2 -19806.861} C_VEL
LIN {X 0,Y 235.215,Z 169.184,A -85,B 0,C 180,E1 -19810.328,E2 -19810.328} C_VEL
LIN {X 0,Y 235.047,Z 169.2,A -85,B 0,C 180,E1 -19815.612,E2 -19815.612} C_VEL
LIN {X 0,Y 234.964,Z 169.217,A -85,B 0,C 180,E1 -19819.21,E2 -19819.21} C_VEL
LIN {X 0,Y 234.936,Z 169.219,A -85,B 0,C 180,E1 -19822.987,E2 -19822.987} C_VEL
LIN {X 0,Y 234.232,Z 169.307,A -85,B 0,C 180,E1 -19824.417,E2 -19824.417} C_VEL
LIN {X 0,Y 231.397,Z 169.661,A -85,B 0,C 180,E1 -19826.752,E2 -19826.752} C_VEL
LIN {X 0,Y 229.001,Z 169.96,A -85,B 0,C 180,E1 -19828.655,E2 -19828.655} C_VEL
LIN {X 0,Y 227.957,Z 170.088,A -85,B 0,C 180,E1 -19830.131,E2 -19830.131} C_VEL
LIN {X 0,Y 227.861,Z 170.099,A -85,B 0,C 180,E1 -19830.631,E2 -19830.631} C_VEL
LIN {X 0,Y 227.881,Z 170.098,A -85,B 0,C 180,E1 -19833.721,E2 -19833.721} C_VEL
LIN {X 0,Y 227.844,Z 170.104,A -85,B 0,C 180,E1 -19838.092,E2 -19838.092} C_VEL
LIN {X 0,Y 227.79,Z 170.115,A -85,B 0,C 180,E1 -19842.748,E2 -19842.748} C_VEL
LIN {X 0,Y 227.796,Z 170.111,A -85,B 0,C 180,E1 -19847.253,E2 -19847.253} C_VEL
LIN {X 0,Y 227.847,Z 170.101,A -85,B 0,C 180,E1 -19851.909,E2 -19851.909} C_VEL
LIN {X 0,Y 227.912,Z 170.238,A -85,B 0,C 180,E1 -19853.656,E2 -19853.656} C_VEL
LIN {X 0,Y 230.109,Z 180.082,A -85,B 0,C 180,E1 -19857.691,E2 -19857.691} C_VEL
LIN {X 0,Y 230.556,Z 182.569,A -85,B 0,C 180,E1 -19858.667,E2 -19858.667} C_VEL
LIN {X 0,Y 236.664,Z 199.831,A -85,B 0,C 180,E1 -19859.946,E2 -19859.946} C_VEL
LIN {X 0,Y 240.916,Z 235.131,A -85,B 0,C 180,E1 -19861.538,E2 -19861.538} C_VEL
LIN {X 0,Y 239.037,Z 291.477,A -85,B 0,C 180,E1 -19863.242,E2 -19863.242} C_VEL
LIN {X 0,Y 238.037,Z 304.617,A -85,B 0,C 180,E1 -19863.948,E2 -19863.948} C_VEL
LIN {X 0,Y 236.684,Z 317.337,A -85,B 0,C 180,E1 -19864.967,E2 -19864.967} C_VEL
LIN {X 0,Y 235.155,Z 328.652,A -85,B 0,C 180,E1 -19866.204,E2 -19866.204} C_VEL
LIN {X 0,Y 233.555,Z 339.067,A -85,B 0,C 180,E1 -19867.672,E2 -19867.672} C_VEL
LIN {X 0,Y 231.832,Z 348.737,A -85,B 0,C 180,E1 -19869.365,E2 -19869.365} C_VEL
LIN {X 0,Y 230.348,Z 357.124,A -85,B 0,C 180,E1 -19871.165,E2 -19871.165} C_VEL
LIN {X 0,Y 229.164,Z 364.45,A -85,B 0,C 180,E1 -19873.061,E2 -19873.061} C_VEL
LIN {X 0,Y 227.723,Z 372.772,A -85,B 0,C 180,E1 -19875.706,E2 -19875.706} C_VEL
LIN {X 0,Y 226.667,Z 379.453,A -85,B 0,C 180,E1 -19878.373,E2 -19878.373} C_VEL
LIN {X 0,Y 226.072,Z 384.765,A -85,B 0,C 180,E1 -19881.057,E2 -19881.057} C_VEL
LIN {X 0,Y 225.761,Z 388.865,A -85,B 0,C 180,E1 -19883.745,E2 -19883.745} C_VEL
LIN {X 0,Y 225.684,Z 391.879,A -85,B 0,C 180,E1 -19886.429,E2 -19886.429} C_VEL
LIN {X 0,Y 225.767,Z 393.342,A -85,B 0,C 180,E1 -19888.216,E2 -19888.216} C_VEL
LIN {X 0,Y 225.821,Z 394.356,A -85,B 0,C 180,E1 -19890,E2 -19890} C_VEL
LIN {X 0,Y 225.738,Z 394.966,A -85,B 0,C 180,E1 -19891.784,E2 -19891.784} C_VEL
LIN {X 0,Y 225.623,Z 395.111,A -85,B 0,C 180,E1 -19894.59,E2 -19894.59} C_VEL
LIN {X 0,Y 225.773,Z 394.406,A -85,B 0,C 180,E1 -19897.152,E2 -19897.152} C_VEL
LIN {X 0,Y 226.599,Z 392.064,A -85,B 0,C 180,E1 -19900.725,E2 -19900.725} C_VEL
LIN {X 0,Y 227.651,Z 389.218,A -85,B 0,C 180,E1 -19903.387,E2 -19903.387} C_VEL
LIN {X 0,Y 229.236,Z 385.379,A -85,B 0,C 180,E1 -19906.017,E2 -19906.017} C_VEL
LIN {X 0,Y 231.404,Z 380.448,A -85,B 0,C 180,E1 -19908.596,E2 -19908.596} C_VEL
LIN {X 0,Y 234.04,Z 373.553,A -85,B 0,C 180,E1 -19911.422,E2 -19911.422} C_VEL
LIN {X 0,Y 237.297,Z 365.184,A -85,B 0,C 180,E1 -19914.031,E2 -19914.031} C_VEL
LIN {X 0,Y 240.308,Z 357.11,A -85,B 0,C 180,E1 -19916.02,E2 -19916.02} C_VEL
LIN {X 0,Y 243.506,Z 347.31,A -85,B 0,C 180,E1 -19917.969,E2 -19917.969} C_VEL
LIN {X 0,Y 246.754,Z 336.359,A -85,B 0,C 180,E1 -19919.661,E2 -19919.661} C_VEL
LIN {X 0,Y 249.869,Z 323.928,A -85,B 0,C 180,E1 -19921.12,E2 -19921.12} C_VEL
LIN {X 0,Y 252.408,Z 311.709,A -85,B 0,C 180,E1 -19922.175,E2 -19922.175} C_VEL
LIN {X 0,Y 254.365,Z 298.858,A -85,B 0,C 180,E1 -19922.953,E2 -19922.953} C_VEL
LIN {X 0,Y 255.524,Z 285.475,A -85,B 0,C 180,E1 -19923.493,E2 -19923.493} C_VEL
LIN {X 0,Y 257.642,Z 239.56,A -85,B 0,C 180,E1 -19924.807,E2 -19924.807} C_VEL
LIN {X 0,Y 255.626,Z 226.14,A -85,B 0,C 180,E1 -19925.713,E2 -19925.713} C_VEL
LIN {X 0,Y 249.662,Z 212.728,A -85,B 0,C 180,E1 -19927.514,E2 -19927.514} C_VEL
LIN {X 0,Y 243.485,Z 200.796,A -85,B 0,C 180,E1 -19929.453,E2 -19929.453} C_VEL
LIN {X 0,Y 237.44,Z 190.593,A -85,B 0,C 180,E1 -19931.46,E2 -19931.46} C_VEL
LIN {X 0,Y 233.988,Z 185.143,A -85,B 0,C 180,E1 -19932.692,E2 -19932.692} C_VEL
LIN {X 0,Y 231.066,Z 180.438,A -85,B 0,C 180,E1 -19933.795,E2 -19933.795} C_VEL
LIN {X 0,Y 229.108,Z 174.309,A -85,B 0,C 180,E1 -19937.556,E2 -19937.556} C_VEL
LIN {X 0,Y 227.83,Z 170.106,A -85,B 0,C 180,E1 -19940.461,E2 -19940.461} C_VEL
LIN {X 0,Y 227.882,Z 170.098,A -85,B 0,C 180,E1 -19944.127,E2 -19944.127} C_VEL
LIN {X 0,Y 227.858,Z 170.093,A -85,B 0,C 180,E1 -19948.375,E2 -19948.375} C_VEL
LIN {X 0,Y 227.846,Z 170.091,A -85,B 0,C 180,E1 -19952.439,E2 -19952.439} C_VEL
LIN {X 0,Y 227.867,Z 170.09,A -85,B 0,C 180,E1 -19956.361,E2 -19956.361} C_VEL
LIN {X 0,Y 227.89,Z 170.096,A -85,B 0,C 180,E1 -19960.169,E2 -19960.169} C_VEL
LIN {X 0,Y 228.011,Z 170.081,A -85,B 0,C 180,E1 -19963.893,E2 -19963.893} C_VEL
LIN {X 0,Y 228.126,Z 170.068,A -85,B 0,C 180,E1 -19969.347,E2 -19969.347} C_VEL
LIN {X 0,Y 228.301,Z 170.034,A -85,B 0,C 180,E1 -19972.926,E2 -19972.926} C_VEL
LIN {X 0,Y 228.538,Z 170.009,A -85,B 0,C 180,E1 -19978.237,E2 -19978.237} C_VEL
LIN {X 0,Y 228.55,Z 170,A -85,B 0,C 180,E1 -19981.761,E2 -19981.761} C_VEL
LIN {X 0,Y 228.308,Z 170.036,A -85,B 0,C 180,E1 -19987.072,E2 -19987.072} C_VEL
LIN {X 0,Y 228.145,Z 170.053,A -85,B 0,C 180,E1 -19990.65,E2 -19990.65} C_VEL
LIN {X 0,Y 228.05,Z 170.067,A -85,B 0,C 180,E1 -19994.272,E2 -19994.272} C_VEL
LIN {X 0,Y 227.997,Z 170.076,A -85,B 0,C 180,E1 -19997.953,E2 -19997.953} C_VEL
LIN {X 0,Y 227.916,Z 170.088,A -85,B 0,C 180,E1 -20002.32,E2 -20002.32} C_VEL
LIN {X 0,Y 227.932,Z 170.088,A -85,B 0,C 180,E1 -20005.206,E2 -20005.206} C_VEL
LIN {X 0,Y 228.858,Z 172.789,A -85,B 0,C 180,E1 -20005.672,E2 -20005.672} C_VEL
LIN {X 0,Y 230.689,Z 174.872,A -85,B 0,C 180,E1 -20006.357,E2 -20006.357} C_VEL
LIN {X 0,Y 231.657,Z 175.775,A -85,B 0,C 180,E1 -20006.7,E2 -20006.7} C_VEL
LIN {X 0,Y 233.711,Z 179.029,A -85,B 0,C 180,E1 -20007.477,E2 -20007.477} C_VEL
LIN {X 0,Y 235.247,Z 180.755,A -85,B 0,C 180,E1 -20008.007,E2 -20008.007} C_VEL
LIN {X 0,Y 241.513,Z 189.878,A -85,B 0,C 180,E1 -20010.13,E2 -20010.13} C_VEL
LIN {X 0,Y 249.003,Z 202.475,A -85,B 0,C 180,E1 -20012.467,E2 -20012.467} C_VEL
LIN {X 0,Y 256.261,Z 216.697,A -85,B 0,C 180,E1 -20014.6,E2 -20014.6} C_VEL
LIN {X 0,Y 258.588,Z 221.947,A -85,B 0,C 180,E1 -20015.269,E2 -20015.269} C_VEL
LIN {X 0,Y 255.843,Z 275.923,A -85,B 0,C 180,E1 -20016.805,E2 -20016.805} C_VEL
LIN {X 0,Y 254.348,Z 289.495,A -85,B 0,C 180,E1 -20017.464,E2 -20017.464} C_VEL
LIN {X 0,Y 252.703,Z 301.078,A -85,B 0,C 180,E1 -20018.332,E2 -20018.332} C_VEL
LIN {X 0,Y 250.38,Z 312.732,A -85,B 0,C 180,E1 -20019.475,E2 -20019.475} C_VEL
LIN {X 0,Y 247.801,Z 323.454,A -85,B 0,C 180,E1 -20020.864,E2 -20020.864} C_VEL
LIN {X 0,Y 244.72,Z 334.12,A -85,B 0,C 180,E1 -20022.616,E2 -20022.616} C_VEL
LIN {X 0,Y 241.482,Z 344.014,A -85,B 0,C 180,E1 -20024.684,E2 -20024.684} C_VEL
LIN {X 0,Y 238.529,Z 351.916,A -85,B 0,C 180,E1 -20026.762,E2 -20026.762} C_VEL
LIN {X 0,Y 235.745,Z 358.788,A -85,B 0,C 180,E1 -20029.015,E2 -20029.015} C_VEL
LIN {X 0,Y 233.104,Z 365.024,A -85,B 0,C 180,E1 -20031.617,E2 -20031.617} C_VEL
LIN {X 0,Y 230.599,Z 370.509,A -85,B 0,C 180,E1 -20034.615,E2 -20034.615} C_VEL
LIN {X 0,Y 228.738,Z 374.318,A -85,B 0,C 180,E1 -20037.474,E2 -20037.474} C_VEL
LIN {X 0,Y 227.337,Z 376.939,A -85,B 0,C 180,E1 -20040.355,E2 -20040.355} C_VEL
LIN {X 0,Y 226.636,Z 378.053,A -85,B 0,C 180,E1 -20042.28,E2 -20042.28} C_VEL
LIN {X 0,Y 226.085,Z 378.749,A -85,B 0,C 180,E1 -20044.351,E2 -20044.351} C_VEL
LIN {X 0,Y 225.734,Z 378.943,A -85,B 0,C 180,E1 -20046.125,E2 -20046.125} C_VEL
LIN {X 0,Y 225.472,Z 378.313,A -85,B 0,C 180,E1 -20049.242,E2 -20049.242} C_VEL
LIN {X 0,Y 225.434,Z 376.877,A -85,B 0,C 180,E1 -20051.835,E2 -20051.835} C_VEL
LIN {X 0,Y 225.752,Z 374.16,A -85,B 0,C 180,E1 -20054.809,E2 -20054.809} C_VEL
LIN {X 0,Y 226.227,Z 370.724,A -85,B 0,C 180,E1 -20057.44,E2 -20057.44} C_VEL
LIN {X 0,Y 226.906,Z 365.976,A -85,B 0,C 180,E1 -20060.192,E2 -20060.192} C_VEL
LIN {X 0,Y 227.944,Z 359.916,A -85,B 0,C 180,E1 -20062.916,E2 -20062.916} C_VEL
LIN {X 0,Y 229.263,Z 352.362,A -85,B 0,C 180,E1 -20065.605,E2 -20065.605} C_VEL
LIN {X 0,Y 230.733,Z 344.632,A -85,B 0,C 180,E1 -20067.818,E2 -20067.818} C_VEL
LIN {X 0,Y 232.433,Z 335.259,A -85,B 0,C 180,E1 -20070,E2 -20070} C_VEL
LIN {X 0,Y 234.172,Z 324.793,A -85,B 0,C 180,E1 -20071.935,E2 -20071.935} C_VEL
LIN {X 0,Y 235.878,Z 313.171,A -85,B 0,C 180,E1 -20073.63,E2 -20073.63} C_VEL
LIN {X 0,Y 237.276,Z 301.069,A -85,B 0,C 180,E1 -20074.992,E2 -20074.992} C_VEL
LIN {X 0,Y 238.481,Z 287.597,A -85,B 0,C 180,E1 -20076.08,E2 -20076.08} C_VEL
LIN {X 0,Y 239.378,Z 274.217,A -85,B 0,C 180,E1 -20076.786,E2 -20076.786} C_VEL
LIN {X 0,Y 241.809,Z 205.538,A -85,B 0,C 180,E1 -20078.823,E2 -20078.823} C_VEL
LIN {X 0,Y 234.086,Z 183.354,A -85,B 0,C 180,E1 -20080.378,E2 -20080.378} C_VEL
LIN {X 0,Y 228.248,Z 170.963,A -85,B 0,C 180,E1 -20081.482,E2 -20081.482} C_VEL
LIN {X 0,Y 228.062,Z 170.078,A -85,B 0,C 180,E1 -20081.583,E2 -20081.583} C_VEL
LIN {X 0,Y 227.994,Z 170.087,A -85,B 0,C 180,E1 -20086.107,E2 -20086.107} C_VEL
LIN {X 0,Y 227.915,Z 170.088,A -85,B 0,C 180,E1 -20091.718,E2 -20091.718} C_VEL
LIN {X 0,Y 227.866,Z 170.071,A -85,B 0,C 180,E1 -20096.566,E2 -20096.566} C_VEL
LIN {X 0,Y 227.867,Z 170.098,A -85,B 0,C 180,E1 -20100.28,E2 -20100.28} C_VEL
LIN {X 0,Y 227.874,Z 170.096,A -85,B 0,C 180,E1 -20103.722,E2 -20103.722} C_VEL
LIN {X 0,Y 227.838,Z 170.097,A -85,B 0,C 180,E1 -20108.093,E2 -20108.093} C_VEL
LIN {X 0,Y 227.784,Z 170.109,A -85,B 0,C 180,E1 -20112.75,E2 -20112.75} C_VEL
LIN {X 0,Y 227.784,Z 170.089,A -85,B 0,C 180,E1 -20117.253,E2 -20117.253} C_VEL
LIN {X 0,Y 227.839,Z 170.101,A -85,B 0,C 180,E1 -20121.909,E2 -20121.909} C_VEL
LIN {X 0,Y 227.878,Z 170.091,A -85,B 0,C 180,E1 -20126.379,E2 -20126.379} C_VEL
LIN {X 0,Y 227.871,Z 170.068,A -85,B 0,C 180,E1 -20130.432,E2 -20130.432} C_VEL
LIN {X 0,Y 227.866,Z 170.09,A -85,B 0,C 180,E1 -20134.419,E2 -20134.419} C_VEL
LIN {X 0,Y 227.92,Z 170.096,A -85,B 0,C 180,E1 -20138.284,E2 -20138.284} C_VEL
LIN {X 0,Y 228.009,Z 170.077,A -85,B 0,C 180,E1 -20143.895,E2 -20143.895} C_VEL
LIN {X 0,Y 228.126,Z 170.065,A -85,B 0,C 180,E1 -20149.349,E2 -20149.349} C_VEL
LIN {X 0,Y 228.302,Z 170.043,A -85,B 0,C 180,E1 -20152.928,E2 -20152.928} C_VEL
LIN {X 0,Y 228.535,Z 170.013,A -85,B 0,C 180,E1 -20158.239,E2 -20158.239} C_VEL
LIN {X 0,Y 228.538,Z 170.015,A -85,B 0,C 180,E1 -20161.763,E2 -20161.763} C_VEL
LIN {X 0,Y 228.304,Z 170.043,A -85,B 0,C 180,E1 -20167.074,E2 -20167.074} C_VEL
LIN {X 0,Y 228.145,Z 170.064,A -85,B 0,C 180,E1 -20170.652,E2 -20170.652} C_VEL
LIN {X 0,Y 228.004,Z 170.076,A -85,B 0,C 180,E1 -20176.107,E2 -20176.107} C_VEL
LIN {X 0,Y 227.929,Z 170.092,A -85,B 0,C 180,E1 -20181.717,E2 -20181.717} C_VEL
LIN {X 0,Y 227.927,Z 170.092,A -85,B 0,C 180,E1 -20186.593,E2 -20186.593} C_VEL
LIN {X 0,Y 227.861,Z 170.099,A -85,B 0,C 180,E1 -20190.631,E2 -20190.631} C_VEL
LIN {X 0,Y 227.16,Z 170.189,A -85,B 0,C 180,E1 -20192.105,E2 -20192.105} C_VEL
LIN {X 0,Y 224.287,Z 170.547,A -85,B 0,C 180,E1 -20194.51,E2 -20194.51} C_VEL
LIN {X 0,Y 221.866,Z 170.849,A -85,B 0,C 180,E1 -20196.473,E2 -20196.473} C_VEL
LIN {X 0,Y 220.834,Z 170.977,A -85,B 0,C 180,E1 -20197.997,E2 -20197.997} C_VEL
LIN {X 0,Y 220.752,Z 170.984,A -85,B 0,C 180,E1 -20198.513,E2 -20198.513} C_VEL
LIN {X 0,Y 220.748,Z 170.993,A -85,B 0,C 180,E1 -20202.923,E2 -20202.923} C_VEL
LIN {X 0,Y 220.754,Z 170.989,A -85,B 0,C 180,E1 -20207.076,E2 -20207.076} C_VEL
LIN {X 0,Y 220.787,Z 170.984,A -85,B 0,C 180,E1 -20210.458,E2 -20210.458} C_VEL
LIN {X 0,Y 220.873,Z 171.143,A -85,B 0,C 180,E1 -20213.087,E2 -20213.087} C_VEL
LIN {X 0,Y 223.249,Z 181.911,A -85,B 0,C 180,E1 -20217.644,E2 -20217.644} C_VEL
LIN {X 0,Y 223.32,Z 182.317,A -85,B 0,C 180,E1 -20217.809,E2 -20217.809} C_VEL
LIN {X 0,Y 230.311,Z 201.8,A -85,B 0,C 180,E1 -20219.324,E2 -20219.324} C_VEL
LIN {X 0,Y 234.315,Z 235.038,A -85,B 0,C 180,E1 -20220.885,E2 -20220.885} C_VEL
LIN {X 0,Y 232.401,Z 291.484,A -85,B 0,C 180,E1 -20222.644,E2 -20222.644} C_VEL
LIN {X 0,Y 231.338,Z 304.72,A -85,B 0,C 180,E1 -20223.377,E2 -20223.377} C_VEL
LIN {X 0,Y 229.95,Z 317.351,A -85,B 0,C 180,E1 -20224.424,E2 -20224.424} C_VEL
LIN {X 0,Y 228.371,Z 328.592,A -85,B 0,C 180,E1 -20225.694,E2 -20225.694} C_VEL
LIN {X 0,Y 226.447,Z 340.273,A -85,B 0,C 180,E1 -20227.413,E2 -20227.413} C_VEL
LIN {X 0,Y 224.791,Z 349.713,A -85,B 0,C 180,E1 -20229.167,E2 -20229.167} C_VEL
LIN {X 0,Y 223.014,Z 359.219,A -85,B 0,C 180,E1 -20231.349,E2 -20231.349} C_VEL
LIN {X 0,Y 221.715,Z 366.555,A -85,B 0,C 180,E1 -20233.424,E2 -20233.424} C_VEL
LIN {X 0,Y 220.556,Z 373.227,A -85,B 0,C 180,E1 -20235.702,E2 -20235.702} C_VEL
LIN {X 0,Y 219.666,Z 378.76,A -85,B 0,C 180,E1 -20237.997,E2 -20237.997} C_VEL
LIN {X 0,Y 219.026,Z 384.161,A -85,B 0,C 180,E1 -20240.767,E2 -20240.767} C_VEL
LIN {X 0,Y 218.698,Z 388.343,A -85,B 0,C 180,E1 -20243.542,E2 -20243.542} C_VEL
LIN {X 0,Y 218.591,Z 391.43,A -85,B 0,C 180,E1 -20246.313,E2 -20246.313} C_VEL
LIN {X 0,Y 218.678,Z 392.954,A -85,B 0,C 180,E1 -20248.158,E2 -20248.158} C_VEL
LIN {X 0,Y 218.754,Z 394.011,A -85,B 0,C 180,E1 -20250,E2 -20250} C_VEL
LIN {X 0,Y 218.649,Z 394.653,A -85,B 0,C 180,E1 -20251.842,E2 -20251.842} C_VEL
LIN {X 0,Y 218.57,Z 394.777,A -85,B 0,C 180,E1 -20255.535,E2 -20255.535} C_VEL
LIN {X 0,Y 219.059,Z 393.29,A -85,B 0,C 180,E1 -20259.231,E2 -20259.231} C_VEL
LIN {X 0,Y 220.3,Z 390.239,A -85,B 0,C 180,E1 -20262.904,E2 -20262.904} C_VEL
LIN {X 0,Y 221.771,Z 386.812,A -85,B 0,C 180,E1 -20265.626,E2 -20265.626} C_VEL
LIN {X 0,Y 223.894,Z 382.339,A -85,B 0,C 180,E1 -20268.294,E2 -20268.294} C_VEL
LIN {X 0,Y 226.762,Z 375.526,A -85,B 0,C 180,E1 -20271.4,E2 -20271.4} C_VEL
LIN {X 0,Y 229.717,Z 368.351,A -85,B 0,C 180,E1 -20273.914,E2 -20273.914} C_VEL
LIN {X 0,Y 233.292,Z 359.355,A -85,B 0,C 180,E1 -20276.382,E2 -20276.382} C_VEL
LIN {X 0,Y 236.983,Z 349.038,A -85,B 0,C 180,E1 -20278.568,E2 -20278.568} C_VEL
LIN {X 0,Y 240.243,Z 338.574,A -85,B 0,C 180,E1 -20280.307,E2 -20280.307} C_VEL
LIN {X 0,Y 243.478,Z 326.931,A -85,B 0,C 180,E1 -20281.788,E2 -20281.788} C_VEL
LIN {X 0,Y 246.277,Z 314.536,A -85,B 0,C 180,E1 -20282.955,E2 -20282.955} C_VEL
LIN {X 0,Y 248.488,Z 301.591,A -85,B 0,C 180,E1 -20283.836,E2 -20283.836} C_VEL
LIN {X 0,Y 249.874,Z 289.22,A -85,B 0,C 180,E1 -20284.402,E2 -20284.402} C_VEL
LIN {X 0,Y 252.318,Z 241.141,A -85,B 0,C 180,E1 -20285.811,E2 -20285.811} C_VEL
LIN {X 0,Y 250.596,Z 229.296,A -85,B 0,C 180,E1 -20286.642,E2 -20286.642} C_VEL
LIN {X 0,Y 245.189,Z 216.894,A -85,B 0,C 180,E1 -20288.361,E2 -20288.361} C_VEL
LIN {X 0,Y 239.333,Z 205.392,A -85,B 0,C 180,E1 -20290.289,E2 -20290.289} C_VEL
LIN {X 0,Y 233.628,Z 195.576,A -85,B 0,C 180,E1 -20292.294,E2 -20292.294} C_VEL
LIN {X 0,Y 230.158,Z 190.042,A -85,B 0,C 180,E1 -20293.591,E2 -20293.591} C_VEL
LIN {X 0,Y 227.008,Z 185.101,A -85,B 0,C 180,E1 -20294.832,E2 -20294.832} C_VEL
LIN {X 0,Y 223.93,Z 180.576,A -85,B 0,C 180,E1 -20296.098,E2 -20296.098} C_VEL
LIN {X 0,Y 223.539,Z 179.701,A -85,B 0,C 180,E1 -20296.312,E2 -20296.312} C_VEL
LIN {X 0,Y 221.626,Z 173.522,A -85,B 0,C 180,E1 -20300.637,E2 -20300.637} C_VEL
LIN {X 0,Y 220.81,Z 170.973,A -85,B 0,C 180,E1 -20302.722,E2 -20302.722} C_VEL
LIN {X 0,Y 220.814,Z 170.98,A -85,B 0,C 180,E1 -20307.242,E2 -20307.242} C_VEL
LIN {X 0,Y 220.8,Z 170.978,A -85,B 0,C 180,E1 -20311.48,E2 -20311.48} C_VEL
LIN {X 0,Y 220.823,Z 170.977,A -85,B 0,C 180,E1 -20315.559,E2 -20315.559} C_VEL
LIN {X 0,Y 220.848,Z 170.974,A -85,B 0,C 180,E1 -20319.509,E2 -20319.509} C_VEL
LIN {X 0,Y 220.972,Z 170.951,A -85,B 0,C 180,E1 -20323.366,E2 -20323.366} C_VEL
LIN {X 0,Y 221.051,Z 170.949,A -85,B 0,C 180,E1 -20329.002,E2 -20329.002} C_VEL
LIN {X 0,Y 221.238,Z 170.912,A -85,B 0,C 180,E1 -20332.699,E2 -20332.699} C_VEL
LIN {X 0,Y 221.471,Z 170.888,A -85,B 0,C 180,E1 -20338.181,E2 -20338.181} C_VEL
LIN {X 0,Y 221.508,Z 170.877,A -85,B 0,C 180,E1 -20341.817,E2 -20341.817} C_VEL
LIN {X 0,Y 221.246,Z 170.918,A -85,B 0,C 180,E1 -20347.299,E2 -20347.299} C_VEL
LIN {X 0,Y 221.067,Z 170.936,A -85,B 0,C 180,E1 -20350.995,E2 -20350.995} C_VEL
LIN {X 0,Y 221.006,Z 170.957,A -85,B 0,C 180,E1 -20356.63,E2 -20356.63} C_VEL
LIN {X 0,Y 220.88,Z 170.972,A -85,B 0,C 180,E1 -20360.486,E2 -20360.486} C_VEL
LIN {X 0,Y 220.858,Z 170.982,A -85,B 0,C 180,E1 -20362.81,E2 -20362.81} C_VEL
LIN {X 0,Y 221.621,Z 173.379,A -85,B 0,C 180,E1 -20363.233,E2 -20363.233} C_VEL
LIN {X 0,Y 223.516,Z 175.671,A -85,B 0,C 180,E1 -20364.04,E2 -20364.04} C_VEL
LIN {X 0,Y 224.783,Z 176.721,A -85,B 0,C 180,E1 -20364.534,E2 -20364.534} C_VEL
LIN {X 0,Y 226.846,Z 179.999,A -85,B 0,C 180,E1 -20365.397,E2 -20365.397} C_VEL
LIN {X 0,Y 228.522,Z 181.779,A -85,B 0,C 180,E1 -20366.029,E2 -20366.029} C_VEL
LIN {X 0,Y 231.006,Z 185.285,A -85,B 0,C 180,E1 -20366.977,E2 -20366.977} C_VEL
LIN {X 0,Y 235.665,Z 191.94,A -85,B 0,C 180,E1 -20368.657,E2 -20368.657} C_VEL
LIN {X 0,Y 240.197,Z 199.097,A -85,B 0,C 180,E1 -20370.203,E2 -20370.203} C_VEL
LIN {X 0,Y 246.677,Z 210.615,A -85,B 0,C 180,E1 -20372.271,E2 -20372.271} C_VEL
LIN {X 0,Y 252.934,Z 223.638,A -85,B 0,C 180,E1 -20374.179,E2 -20374.179} C_VEL
LIN {X 0,Y 253.27,Z 224.995,A -85,B 0,C 180,E1 -20374.303,E2 -20374.303} C_VEL
LIN {X 0,Y 250.347,Z 277.075,A -85,B 0,C 180,E1 -20375.802,E2 -20375.802} C_VEL
LIN {X 0,Y 248.755,Z 290.685,A -85,B 0,C 180,E1 -20376.492,E2 -20376.492} C_VEL
LIN {X 0,Y 246.858,Z 303.14,A -85,B 0,C 180,E1 -20377.477,E2 -20377.477} C_VEL
LIN {X 0,Y 244.284,Z 314.878,A -85,B 0,C 180,E1 -20378.705,E2 -20378.705} C_VEL
LIN {X 0,Y 241.259,Z 326.584,A -85,B 0,C 180,E1 -20380.329,E2 -20380.329} C_VEL
LIN {X 0,Y 238.067,Z 336.739,A -85,B 0,C 180,E1 -20382.122,E2 -20382.122} C_VEL
LIN {X 0,Y 234.906,Z 345.619,A -85,B 0,C 180,E1 -20384.107,E2 -20384.107} C_VEL
LIN {X 0,Y 231.533,Z 354.123,A -85,B 0,C 180,E1 -20386.501,E2 -20386.501} C_VEL
LIN {X 0,Y 228.341,Z 361.496,A -85,B 0,C 180,E1 -20389.153,E2 -20389.153} C_VEL
LIN {X 0,Y 225.961,Z 366.66,A -85,B 0,C 180,E1 -20391.534,E2 -20391.534} C_VEL
LIN {X 0,Y 223.659,Z 371.335,A -85,B 0,C 180,E1 -20394.299,E2 -20394.299} C_VEL
LIN {X 0,Y 221.646,Z 375.107,A -85,B 0,C 180,E1 -20397.382,E2 -20397.382} C_VEL
LIN {X 0,Y 220.678,Z 376.837,A -85,B 0,C 180,E1 -20399.366,E2 -20399.366} C_VEL
LIN {X 0,Y 219.833,Z 378.108,A -85,B 0,C 180,E1 -20401.344,E2 -20401.344} C_VEL
LIN {X 0,Y 219.077,Z 379.006,A -85,B 0,C 180,E1 -20403.925,E2 -20403.925} C_VEL
LIN {X 0,Y 218.498,Z 379.064,A -85,B 0,C 180,E1 -20407.296,E2 -20407.296} C_VEL
LIN {X 0,Y 218.384,Z 378.461,A -85,B 0,C 180,E1 -20409.268,E2 -20409.268} C_VEL
LIN {X 0,Y 218.32,Z 377.432,A -85,B 0,C 180,E1 -20411.222,E2 -20411.222} C_VEL
LIN {X 0,Y 218.627,Z 374.531,A -85,B 0,C 180,E1 -20414.658,E2 -20414.658} C_VEL
LIN {X 0,Y 219.25,Z 370.219,A -85,B 0,C 180,E1 -20417.974,E2 -20417.974} C_VEL
LIN {X 0,Y 220.013,Z 365.252,A -85,B 0,C 180,E1 -20420.81,E2 -20420.81} C_VEL
LIN {X 0,Y 221.117,Z 358.972,A -85,B 0,C 180,E1 -20423.613,E2 -20423.613} C_VEL
LIN {X 0,Y 222.527,Z 351.16,A -85,B 0,C 180,E1 -20426.379,E2 -20426.379} C_VEL
LIN {X 0,Y 224.124,Z 342.946,A -85,B 0,C 180,E1 -20428.691,E2 -20428.691} C_VEL
LIN {X 0,Y 225.981,Z 333.234,A -85,B 0,C 180,E1 -20430.891,E2 -20430.891} C_VEL
LIN {X 0,Y 227.759,Z 322.311,A -85,B 0,C 180,E1 -20432.875,E2 -20432.875} C_VEL
LIN {X 0,Y 229.387,Z 311.62,A -85,B 0,C 180,E1 -20434.393,E2 -20434.393} C_VEL
LIN {X 0,Y 230.737,Z 299.961,A -85,B 0,C 180,E1 -20435.681,E2 -20435.681} C_VEL
LIN {X 0,Y 231.898,Z 286.816,A -85,B 0,C 180,E1 -20436.745,E2 -20436.745} C_VEL
LIN {X 0,Y 232.801,Z 273.599,A -85,B 0,C 180,E1 -20437.426,E2 -20437.426} C_VEL
LIN {X 0,Y 235.257,Z 207.212,A -85,B 0,C 180,E1 -20439.439,E2 -20439.439} C_VEL
LIN {X 0,Y 228.157,Z 186.49,A -85,B 0,C 180,E1 -20440.943,E2 -20440.943} C_VEL
LIN {X 0,Y 221.175,Z 171.906,A -85,B 0,C 180,E1 -20442.315,E2 -20442.315} C_VEL
LIN {X 0,Y 220.98,Z 170.96,A -85,B 0,C 180,E1 -20442.443,E2 -20442.443} C_VEL
LIN {X 0,Y 220.911,Z 170.968,A -85,B 0,C 180,E1 -20447.371,E2 -20447.371} C_VEL
LIN {X 0,Y 220.851,Z 170.963,A -85,B 0,C 180,E1 -20452.45,E2 -20452.45} C_VEL
LIN {X 0,Y 220.822,Z 170.95,A -85,B 0,C 180,E1 -20456.985,E2 -20456.985} C_VEL
LIN {X 0,Y 220.816,Z 170.977,A -85,B 0,C 180,E1 -20460.76,E2 -20460.76} C_VEL
LIN {X 0,Y 220.791,Z 170.971,A -85,B 0,C 180,E1 -20464.957,E2 -20464.957} C_VEL
LIN {X 0,Y 220.799,Z 170.968,A -85,B 0,C 180,E1 -20467.276,E2 -20467.276} C_VEL
LIN {X 0,Y 220.746,Z 170.985,A -85,B 0,C 180,E1 -20471.959,E2 -20471.959} C_VEL
LIN {X 0,Y 220.751,Z 170.967,A -85,B 0,C 180,E1 -20475.542,E2 -20475.542} C_VEL
LIN {X 0,Y 220.78,Z 170.976,A -85,B 0,C 180,E1 -20480.459,E2 -20480.459} C_VEL
LIN {X 0,Y 220.824,Z 170.979,A -85,B 0,C 180,E1 -20482.794,E2 -20482.794} C_VEL
LIN {X 0,Y 220.811,Z 170.964,A -85,B 0,C 180,E1 -20487.244,E2 -20487.244} C_VEL
LIN {X 0,Y 220.795,Z 170.951,A -85,B 0,C 180,E1 -20491.482,E2 -20491.482} C_VEL
LIN {X 0,Y 220.797,Z 170.975,A -85,B 0,C 180,E1 -20495.558,E2 -20495.558} C_VEL
LIN {X 0,Y 220.847,Z 170.974,A -85,B 0,C 180,E1 -20499.511,E2 -20499.511} C_VEL
LIN {X 0,Y 220.971,Z 170.951,A -85,B 0,C 180,E1 -20503.368,E2 -20503.368} C_VEL
LIN {X 0,Y 221.048,Z 170.946,A -85,B 0,C 180,E1 -20509.004,E2 -20509.004} C_VEL
LIN {X 0,Y 221.239,Z 170.923,A -85,B 0,C 180,E1 -20512.701,E2 -20512.701} C_VEL
LIN {X 0,Y 221.469,Z 170.893,A -85,B 0,C 180,E1 -20518.182,E2 -20518.182} C_VEL
LIN {X 0,Y 221.471,Z 170.896,A -85,B 0,C 180,E1 -20521.819,E2 -20521.819} C_VEL
LIN {X 0,Y 221.242,Z 170.921,A -85,B 0,C 180,E1 -20527.301,E2 -20527.301} C_VEL
LIN {X 0,Y 221.064,Z 170.947,A -85,B 0,C 180,E1 -20530.998,E2 -20530.998} C_VEL
LIN {X 0,Y 220.97,Z 170.951,A -85,B 0,C 180,E1 -20536.634,E2 -20536.634} C_VEL
LIN {X 0,Y 220.854,Z 170.973,A -85,B 0,C 180,E1 -20540.491,E2 -20540.491} C_VEL
LIN {X 0,Y 220.849,Z 170.974,A -85,B 0,C 180,E1 -20544.438,E2 -20544.438} C_VEL
LIN {X 0,Y 220.808,Z 170.979,A -85,B 0,C 180,E1 -20548.519,E2 -20548.519} C_VEL
LIN {X 0,Y 220.816,Z 170.98,A -85,B 0,C 180,E1 -20552.757,E2 -20552.757} C_VEL
LIN {X 0,Y 220.806,Z 170.982,A -85,B 0,C 180,E1 -20557.276,E2 -20557.276} C_VEL
LIN {X 0,Y 220.752,Z 170.984,A -85,B 0,C 180,E1 -20558.513,E2 -20558.513} C_VEL
LIN {X 0,Y 220.101,Z 171.071,A -85,B 0,C 180,E1 -20560.037,E2 -20560.037} C_VEL
LIN {X 0,Y 217.294,Z 171.428,A -85,B 0,C 180,E1 -20562.525,E2 -20562.525} C_VEL
LIN {X 0,Y 214.042,Z 171.831,A -85,B 0,C 180,E1 -20565.6,E2 -20565.6} C_VEL
LIN {X 0,Y 213.682,Z 171.869,A -85,B 0,C 180,E1 -20566.666,E2 -20566.666} C_VEL
LIN {X 0,Y 213.712,Z 171.863,A -85,B 0,C 180,E1 -20571.33,E2 -20571.33} C_VEL
LIN {X 0,Y 213.755,Z 171.935,A -85,B 0,C 180,E1 -20572.424,E2 -20572.424} C_VEL
LIN {X 0,Y 215.793,Z 180.889,A -85,B 0,C 180,E1 -20576.381,E2 -20576.381} C_VEL
LIN {X 0,Y 216.089,Z 182.188,A -85,B 0,C 180,E1 -20576.889,E2 -20576.889} C_VEL
LIN {X 0,Y 223.915,Z 203.593,A -85,B 0,C 180,E1 -20578.654,E2 -20578.654} C_VEL
LIN {X 0,Y 227.771,Z 236.476,A -85,B 0,C 180,E1 -20580.25,E2 -20580.25} C_VEL
LIN {X 0,Y 225.764,Z 291.652,A -85,B 0,C 180,E1 -20582.018,E2 -20582.018} C_VEL
LIN {X 0,Y 224.613,Z 305.567,A -85,B 0,C 180,E1 -20582.83,E2 -20582.83} C_VEL
LIN {X 0,Y 223.108,Z 318.355,A -85,B 0,C 180,E1 -20583.957,E2 -20583.957} C_VEL
LIN {X 0,Y 221.389,Z 330.117,A -85,B 0,C 180,E1 -20585.376,E2 -20585.376} C_VEL
LIN {X 0,Y 219.342,Z 341.455,A -85,B 0,C 180,E1 -20587.138,E2 -20587.138} C_VEL
LIN {X 0,Y 217.595,Z 351.699,A -85,B 0,C 180,E1 -20589.189,E2 -20589.189} C_VEL
LIN {X 0,Y 216.035,Z 359.221,A -85,B 0,C 180,E1 -20591.015,E2 -20591.015} C_VEL
LIN {X 0,Y 214.598,Z 367.114,A -85,B 0,C 180,E1 -20593.347,E2 -20593.347} C_VEL
LIN {X 0,Y 213.197,Z 374.792,A -85,B 0,C 180,E1 -20596.172,E2 -20596.172} C_VEL
LIN {X 0,Y 212.164,Z 381.873,A -85,B 0,C 180,E1 -20599.502,E2 -20599.502} C_VEL
LIN {X 0,Y 211.7,Z 386.534,A -85,B 0,C 180,E1 -20602.369,E2 -20602.369} C_VEL
LIN {X 0,Y 211.476,Z 390.386,A -85,B 0,C 180,E1 -20605.568,E2 -20605.568} C_VEL
LIN {X 0,Y 211.59,Z 392.536,A -85,B 0,C 180,E1 -20608.096,E2 -20608.096} C_VEL
LIN {X 0,Y 211.688,Z 393.663,A -85,B 0,C 180,E1 -20610,E2 -20610} C_VEL
LIN {X 0,Y 211.56,Z 394.339,A -85,B 0,C 180,E1 -20611.903,E2 -20611.903} C_VEL
LIN {X 0,Y 211.49,Z 394.534,A -85,B 0,C 180,E1 -20615.721,E2 -20615.721} C_VEL
LIN {X 0,Y 211.641,Z 394.054,A -85,B 0,C 180,E1 -20617.633,E2 -20617.633} C_VEL
LIN {X 0,Y 212.619,Z 391.86,A -85,B 0,C 180,E1 -20621.439,E2 -20621.439} C_VEL
LIN {X 0,Y 213.786,Z 389.164,A -85,B 0,C 180,E1 -20624.274,E2 -20624.274} C_VEL
LIN {X 0,Y 215.605,Z 385.483,A -85,B 0,C 180,E1 -20627.06,E2 -20627.06} C_VEL
LIN {X 0,Y 217.931,Z 380.72,A -85,B 0,C 180,E1 -20629.792,E2 -20629.792} C_VEL
LIN {X 0,Y 221.056,Z 373.626,A -85,B 0,C 180,E1 -20632.921,E2 -20632.921} C_VEL
LIN {X 0,Y 224.434,Z 365.959,A -85,B 0,C 180,E1 -20635.504,E2 -20635.504} C_VEL
LIN {X 0,Y 227.681,Z 358.161,A -85,B 0,C 180,E1 -20637.582,E2 -20637.582} C_VEL
LIN {X 0,Y 231.553,Z 347.629,A -85,B 0,C 180,E1 -20639.802,E2 -20639.802} C_VEL
LIN {X 0,Y 234.612,Z 338.228,A -85,B 0,C 180,E1 -20641.364,E2 -20641.364} C_VEL
LIN {X 0,Y 237.961,Z 326.589,A -85,B 0,C 180,E1 -20642.867,E2 -20642.867} C_VEL
LIN {X 0,Y 240.853,Z 314.19,A -85,B 0,C 180,E1 -20644.048,E2 -20644.048} C_VEL
LIN {X 0,Y 243.033,Z 301.96,A -85,B 0,C 180,E1 -20644.892,E2 -20644.892} C_VEL
LIN {X 0,Y 244.596,Z 288.891,A -85,B 0,C 180,E1 -20645.498,E2 -20645.498} C_VEL
LIN {X 0,Y 247.062,Z 242.066,A -85,B 0,C 180,E1 -20646.895,E2 -20646.895} C_VEL
LIN {X 0,Y 245.606,Z 232.183,A -85,B 0,C 180,E1 -20647.626,E2 -20647.626} C_VEL
LIN {X 0,Y 240.77,Z 221.054,A -85,B 0,C 180,E1 -20649.239,E2 -20649.239} C_VEL
LIN {X 0,Y 235.325,Z 210.15,A -85,B 0,C 180,E1 -20651.13,E2 -20651.13} C_VEL
LIN {X 0,Y 229.779,Z 200.342,A -85,B 0,C 180,E1 -20653.192,E2 -20653.192} C_VEL
LIN {X 0,Y 226.521,Z 195.062,A -85,B 0,C 180,E1 -20654.471,E2 -20654.471} C_VEL
LIN {X 0,Y 223.551,Z 190.391,A -85,B 0,C 180,E1 -20655.695,E2 -20655.695} C_VEL
LIN {X 0,Y 219.874,Z 184.883,A -85,B 0,C 180,E1 -20657.297,E2 -20657.297} C_VEL
LIN {X 0,Y 216.712,Z 180.388,A -85,B 0,C 180,E1 -20658.785,E2 -20658.785} C_VEL
LIN {X 0,Y 216.066,Z 179.114,A -85,B 0,C 180,E1 -20659.201,E2 -20659.201} C_VEL
LIN {X 0,Y 214.779,Z 174.975,A -85,B 0,C 180,E1 -20662.408,E2 -20662.408} C_VEL
LIN {X 0,Y 213.764,Z 171.848,A -85,B 0,C 180,E1 -20665.145,E2 -20665.145} C_VEL
LIN {X 0,Y 213.77,Z 171.845,A -85,B 0,C 180,E1 -20668.736,E2 -20668.736} C_VEL
LIN {X 0,Y 213.785,Z 171.841,A -85,B 0,C 180,E1 -20672.597,E2 -20672.597} C_VEL
LIN {X 0,Y 213.797,Z 171.838,A -85,B 0,C 180,E1 -20676.988,E2 -20676.988} C_VEL
LIN {X 0,Y 213.88,Z 171.829,A -85,B 0,C 180,E1 -20682.797,E2 -20682.797} C_VEL
LIN {X 0,Y 213.916,Z 171.822,A -85,B 0,C 180,E1 -20686.703,E2 -20686.703} C_VEL
LIN {X 0,Y 214.129,Z 171.801,A -85,B 0,C 180,E1 -20690.554,E2 -20690.554} C_VEL
LIN {X 0,Y 214.077,Z 171.817,A -85,B 0,C 180,E1 -20694.347,E2 -20694.347} C_VEL
LIN {X 0,Y 214.408,Z 171.766,A -85,B 0,C 180,E1 -20698.121,E2 -20698.121} C_VEL
LIN {X 0,Y 214.516,Z 171.755,A -85,B 0,C 180,E1 -20699.999,E2 -20699.999} C_VEL
LIN {X 0,Y 214.441,Z 171.757,A -85,B 0,C 180,E1 -20701.877,E2 -20701.877} C_VEL
LIN {X 0,Y 214.187,Z 171.799,A -85,B 0,C 180,E1 -20707.541,E2 -20707.541} C_VEL
LIN {X 0,Y 213.998,Z 171.818,A -85,B 0,C 180,E1 -20711.363,E2 -20711.363} C_VEL
LIN {X 0,Y 213.92,Z 171.828,A -85,B 0,C 180,E1 -20715.237,E2 -20715.237} C_VEL
LIN {X 0,Y 213.831,Z 171.842,A -85,B 0,C 180,E1 -20719.187,E2 -20719.187} C_VEL
LIN {X 0,Y 213.83,Z 171.85,A -85,B 0,C 180,E1 -20719.999,E2 -20719.999} C_VEL
LIN {X 0,Y 214.757,Z 174.579,A -85,B 0,C 180,E1 -20720.596,E2 -20720.596} C_VEL
LIN {X 0,Y 216.682,Z 176.724,A -85,B 0,C 180,E1 -20721.524,E2 -20721.524} C_VEL
LIN {X 0,Y 217.908,Z 177.593,A -85,B 0,C 180,E1 -20722.065,E2 -20722.065} C_VEL
LIN {X 0,Y 219.817,Z 180.792,A -85,B 0,C 180,E1 -20722.989,E2 -20722.989} C_VEL
LIN {X 0,Y 221.899,Z 182.988,A -85,B 0,C 180,E1 -20723.878,E2 -20723.878} C_VEL
LIN {X 0,Y 224.502,Z 186.541,A -85,B 0,C 180,E1 -20724.968,E2 -20724.968} C_VEL
LIN {X 0,Y 226.105,Z 188.746,A -85,B 0,C 180,E1 -20725.614,E2 -20725.614} C_VEL
LIN {X 0,Y 229.374,Z 193.248,A -85,B 0,C 180,E1 -20726.878,E2 -20726.878} C_VEL
LIN {X 0,Y 234.209,Z 200.406,A -85,B 0,C 180,E1 -20728.649,E2 -20728.649} C_VEL
LIN {X 0,Y 241.412,Z 213.152,A -85,B 0,C 180,E1 -20731.125,E2 -20731.125} C_VEL
LIN {X 0,Y 247.841,Z 226.467,A -85,B 0,C 180,E1 -20733.189,E2 -20733.189} C_VEL
LIN {X 0,Y 247.722,Z 231.51,A -85,B 0,C 180,E1 -20733.369,E2 -20733.369} C_VEL
LIN {X 0,Y 245.062,Z 277.174,A -85,B 0,C 180,E1 -20734.708,E2 -20734.708} C_VEL
LIN {X 0,Y 243.362,Z 291.155,A -85,B 0,C 180,E1 -20735.424,E2 -20735.424} C_VEL
LIN {X 0,Y 241.338,Z 303.745,A -85,B 0,C 180,E1 -20736.441,E2 -20736.441} C_VEL
LIN {X 0,Y 238.465,Z 316.226,A -85,B 0,C 180,E1 -20737.786,E2 -20737.786} C_VEL
LIN {X 0,Y 235.371,Z 327.555,A -85,B 0,C 180,E1 -20739.411,E2 -20739.411} C_VEL
LIN {X 0,Y 231.966,Z 337.732,A -85,B 0,C 180,E1 -20741.277,E2 -20741.277} C_VEL
LIN {X 0,Y 228.871,Z 345.978,A -85,B 0,C 180,E1 -20743.172,E2 -20743.172} C_VEL
LIN {X 0,Y 225.688,Z 353.624,A -85,B 0,C 180,E1 -20745.35,E2 -20745.35} C_VEL
LIN {X 0,Y 222.493,Z 360.6,A -85,B 0,C 180,E1 -20747.838,E2 -20747.838} C_VEL
LIN {X 0,Y 219.905,Z 365.983,A -85,B 0,C 180,E1 -20750.269,E2 -20750.269} C_VEL
LIN {X 0,Y 217.267,Z 371.089,A -85,B 0,C 180,E1 -20753.244,E2 -20753.244} C_VEL
LIN {X 0,Y 215.156,Z 374.885,A -85,B 0,C 180,E1 -20756.269,E2 -20756.269} C_VEL
LIN {X 0,Y 213.855,Z 377.024,A -85,B 0,C 180,E1 -20758.697,E2 -20758.697} C_VEL
LIN {X 0,Y 212.392,Z 379.004,A -85,B 0,C 180,E1 -20762.403,E2 -20762.403} C_VEL
LIN {X 0,Y 211.844,Z 379.411,A -85,B 0,C 180,E1 -20764.451,E2 -20764.451} C_VEL
LIN {X 0,Y 211.483,Z 379.381,A -85,B 0,C 180,E1 -20766.498,E2 -20766.498} C_VEL
LIN {X 0,Y 211.321,Z 378.898,A -85,B 0,C 180,E1 -20768.621,E2 -20768.621} C_VEL
LIN {X 0,Y 211.217,Z 377.988,A -85,B 0,C 180,E1 -20770.565,E2 -20770.565} C_VEL
LIN {X 0,Y 211.294,Z 376.614,A -85,B 0,C 180,E1 -20772.581,E2 -20772.581} C_VEL
LIN {X 0,Y 211.677,Z 373.698,A -85,B 0,C 180,E1 -20775.581,E2 -20775.581} C_VEL
LIN {X 0,Y 212.28,Z 369.702,A -85,B 0,C 180,E1 -20778.543,E2 -20778.543} C_VEL
LIN {X 0,Y 213.153,Z 364.38,A -85,B 0,C 180,E1 -20781.544,E2 -20781.544} C_VEL
LIN {X 0,Y 214.297,Z 358.014,A -85,B 0,C 180,E1 -20784.354,E2 -20784.354} C_VEL
LIN {X 0,Y 215.875,Z 349.825,A -85,B 0,C 180,E1 -20787.201,E2 -20787.201} C_VEL
LIN {X 0,Y 217.538,Z 341.279,A -85,B 0,C 180,E1 -20789.584,E2 -20789.584} C_VEL
LIN {X 0,Y 219.5,Z 331.208,A -85,B 0,C 180,E1 -20791.835,E2 -20791.835} C_VEL
LIN {X 0,Y 221.2,Z 321.04,A -85,B 0,C 180,E1 -20793.644,E2 -20793.644} C_VEL
LIN {X 0,Y 222.883,Z 309.941,A -85,B 0,C 180,E1 -20795.202,E2 -20795.202} C_VEL
LIN {X 0,Y 224.345,Z 297.723,A -85,B 0,C 180,E1 -20796.521,E2 -20796.521} C_VEL
LIN {X 0,Y 225.439,Z 285.107,A -85,B 0,C 180,E1 -20797.501,E2 -20797.501} C_VEL
LIN {X 0,Y 226.318,Z 271.794,A -85,B 0,C 180,E1 -20798.146,E2 -20798.146} C_VEL
LIN {X 0,Y 228.647,Z 208.239,A -85,B 0,C 180,E1 -20800.122,E2 -20800.122} C_VEL
LIN {X 0,Y 222.158,Z 189.451,A -85,B 0,C 180,E1 -20801.555,E2 -20801.555} C_VEL
LIN {X 0,Y 214.719,Z 174.386,A -85,B 0,C 180,E1 -20803.068,E2 -20803.068} C_VEL
LIN {X 0,Y 213.898,Z 171.844,A -85,B 0,C 180,E1 -20803.297,E2 -20803.297} C_VEL
LIN {X 0,Y 213.848,Z 171.849,A -85,B 0,C 180,E1 -20807.626,E2 -20807.626} C_VEL
LIN {X 0,Y 213.776,Z 171.834,A -85,B 0,C 180,E1 -20813.001,E2 -20813.001} C_VEL
LIN {X 0,Y 213.764,Z 171.83,A -85,B 0,C 180,E1 -20817.418,E2 -20817.418} C_VEL
LIN {X 0,Y 213.756,Z 171.859,A -85,B 0,C 180,E1 -20821.74,E2 -20821.74} C_VEL
LIN {X 0,Y 213.739,Z 171.842,A -85,B 0,C 180,E1 -20826.29,E2 -20826.29} C_VEL
LIN {X 0,Y 213.696,Z 171.867,A -85,B 0,C 180,E1 -20831.13,E2 -20831.13} C_VEL
LIN {X 0,Y 213.7,Z 171.857,A -85,B 0,C 180,E1 -20833.681,E2 -20833.681} C_VEL
LIN {X 0,Y 213.7,Z 171.84,A -85,B 0,C 180,E1 -20836.347,E2 -20836.347} C_VEL
LIN {X 0,Y 213.704,Z 171.862,A -85,B 0,C 180,E1 -20841.331,E2 -20841.331} C_VEL
LIN {X 0,Y 213.754,Z 171.852,A -85,B 0,C 180,E1 -20846.019,E2 -20846.019} C_VEL
LIN {X 0,Y 213.747,Z 171.823,A -85,B 0,C 180,E1 -20850.45,E2 -20850.45} C_VEL
LIN {X 0,Y 213.747,Z 171.849,A -85,B 0,C 180,E1 -20854.696,E2 -20854.696} C_VEL
LIN {X 0,Y 213.776,Z 171.856,A -85,B 0,C 180,E1 -20858.801,E2 -20858.801} C_VEL
LIN {X 0,Y 213.88,Z 171.834,A -85,B 0,C 180,E1 -20862.799,E2 -20862.799} C_VEL
LIN {X 0,Y 213.905,Z 171.84,A -85,B 0,C 180,E1 -20866.705,E2 -20866.705} C_VEL
LIN {X 0,Y 214.131,Z 171.802,A -85,B 0,C 180,E1 -20870.556,E2 -20870.556} C_VEL
LIN {X 0,Y 214.074,Z 171.82,A -85,B 0,C 180,E1 -20874.349,E2 -20874.349} C_VEL
LIN {X 0,Y 214.405,Z 171.773,A -85,B 0,C 180,E1 -20878.123,E2 -20878.123} C_VEL
LIN {X 0,Y 214.515,Z 171.756,A -85,B 0,C 180,E1 -20880.001,E2 -20880.001} C_VEL
LIN {X 0,Y 214.408,Z 171.776,A -85,B 0,C 180,E1 -20881.879,E2 -20881.879} C_VEL
LIN {X 0,Y 214.184,Z 171.798,A -85,B 0,C 180,E1 -20887.543,E2 -20887.543} C_VEL
LIN {X 0,Y 213.993,Z 171.83,A -85,B 0,C 180,E1 -20891.366,E2 -20891.366} C_VEL
LIN {X 0,Y 213.873,Z 171.838,A -85,B 0,C 180,E1 -20895.242,E2 -20895.242} C_VEL
LIN {X 0,Y 213.796,Z 171.854,A -85,B 0,C 180,E1 -20899.192,E2 -20899.192} C_VEL
LIN {X 0,Y 213.798,Z 171.855,A -85,B 0,C 180,E1 -20903.234,E2 -20903.234} C_VEL
LIN {X 0,Y 213.791,Z 171.854,A -85,B 0,C 180,E1 -20907.428,E2 -20907.428} C_VEL
LIN {X 0,Y 213.763,Z 171.857,A -85,B 0,C 180,E1 -20911.739,E2 -20911.739} C_VEL
LIN {X 0,Y 213.746,Z 171.86,A -85,B 0,C 180,E1 -20916.289,E2 -20916.289} C_VEL
LIN {X 0,Y 213.702,Z 171.87,A -85,B 0,C 180,E1 -20921.129,E2 -20921.129} C_VEL
LIN {X 0,Y 213.705,Z 171.867,A -85,B 0,C 180,E1 -20923.68,E2 -20923.68} C_VEL
LIN {X 0,Y 213.682,Z 171.869,A -85,B 0,C 180,E1 -20926.666,E2 -20926.666} C_VEL
LIN {X 0,Y 212.906,Z 172.02,A -85,B 0,C 180,E1 -20927.752,E2 -20927.752} C_VEL
LIN {X 0,Y 207.231,Z 172.705,A -85,B 0,C 180,E1 -20931.145,E2 -20931.145} C_VEL
LIN {X 0,Y 206.836,Z 173.339,A -85,B 0,C 180,E1 -20931.992,E2 -20931.992} C_VEL
LIN {X 0,Y 206.889,Z 173.617,A -85,B 0,C 180,E1 -20932.146,E2 -20932.146} C_VEL
LIN {X 0,Y 208.743,Z 181.72,A -85,B 0,C 180,E1 -20935.861,E2 -20935.861} C_VEL
LIN {X 0,Y 216.825,Z 203.18,A -85,B 0,C 180,E1 -20937.771,E2 -20937.771} C_VEL
LIN {X 0,Y 217.813,Z 206.983,A -85,B 0,C 180,E1 -20938.037,E2 -20938.037} C_VEL
LIN {X 0,Y 221.227,Z 236.152,A -85,B 0,C 180,E1 -20939.511,E2 -20939.511} C_VEL
LIN {X 0,Y 219.207,Z 291.098,A -85,B 0,C 180,E1 -20941.32,E2 -20941.32} C_VEL
LIN {X 0,Y 218.017,Z 304.868,A -85,B 0,C 180,E1 -20942.132,E2 -20942.132} C_VEL
LIN {X 0,Y 216.527,Z 317.299,A -85,B 0,C 180,E1 -20943.233,E2 -20943.233} C_VEL
LIN {X 0,Y 214.866,Z 328.427,A -85,B 0,C 180,E1 -20944.576,E2 -20944.576} C_VEL
LIN {X 0,Y 212.825,Z 340.047,A -85,B 0,C 180,E1 -20946.396,E2 -20946.396} C_VEL
LIN {X 0,Y 211.044,Z 349.436,A -85,B 0,C 180,E1 -20948.255,E2 -20948.255} C_VEL
LIN {X 0,Y 209.198,Z 358.151,A -85,B 0,C 180,E1 -20950.369,E2 -20950.369} C_VEL
LIN {X 0,Y 208.068,Z 364.702,A -85,B 0,C 180,E1 -20952.302,E2 -20952.302} C_VEL
LIN {X 0,Y 206.502,Z 372.85,A -85,B 0,C 180,E1 -20955.211,E2 -20955.211} C_VEL
LIN {X 0,Y 205.396,Z 379.366,A -85,B 0,C 180,E1 -20958.152,E2 -20958.152} C_VEL
LIN {X 0,Y 204.784,Z 384.516,A -85,B 0,C 180,E1 -20961.115,E2 -20961.115} C_VEL
LIN {X 0,Y 204.494,Z 388.486,A -85,B 0,C 180,E1 -20964.082,E2 -20964.082} C_VEL
LIN {X 0,Y 204.408,Z 390.511,A -85,B 0,C 180,E1 -20966.057,E2 -20966.057} C_VEL
LIN {X 0,Y 204.504,Z 392.115,A -85,B 0,C 180,E1 -20968.03,E2 -20968.03} C_VEL
LIN {X 0,Y 204.599,Z 393.301,A -85,B 0,C 180,E1 -20970,E2 -20970} C_VEL
LIN {X 0,Y 204.473,Z 394.025,A -85,B 0,C 180,E1 -20971.969,E2 -20971.969} C_VEL
LIN {X 0,Y 204.398,Z 394.289,A -85,B 0,C 180,E1 -20975.92,E2 -20975.92} C_VEL
LIN {X 0,Y 204.604,Z 393.853,A -85,B 0,C 180,E1 -20977.897,E2 -20977.897} C_VEL
LIN {X 0,Y 205.006,Z 393.014,A -85,B 0,C 180,E1 -20979.869,E2 -20979.869} C_VEL
LIN {X 0,Y 206.395,Z 390.109,A -85,B 0,C 180,E1 -20983.789,E2 -20983.789} C_VEL
LIN {X 0,Y 208.119,Z 386.836,A -85,B 0,C 180,E1 -20986.68,E2 -20986.68} C_VEL
LIN {X 0,Y 210.403,Z 382.531,A -85,B 0,C 180,E1 -20989.513,E2 -20989.513} C_VEL
LIN {X 0,Y 213.257,Z 376.701,A -85,B 0,C 180,E1 -20992.466,E2 -20992.466} C_VEL
LIN {X 0,Y 216.221,Z 370.323,A -85,B 0,C 180,E1 -20994.995,E2 -20994.995} C_VEL
LIN {X 0,Y 220.027,Z 361.952,A -85,B 0,C 180,E1 -20997.591,E2 -20997.591} C_VEL
LIN {X 0,Y 223.586,Z 353.368,A -85,B 0,C 180,E1 -20999.674,E2 -20999.674} C_VEL
LIN {X 0,Y 227.341,Z 342.858,A -85,B 0,C 180,E1 -21001.704,E2 -21001.704} C_VEL
LIN {X 0,Y 230.761,Z 332.438,A -85,B 0,C 180,E1 -21003.244,E2 -21003.244} C_VEL
LIN {X 0,Y 233.914,Z 320.98,A -85,B 0,C 180,E1 -21004.548,E2 -21004.548} C_VEL
LIN {X 0,Y 236.68,Z 307.905,A -85,B 0,C 180,E1 -21005.644,E2 -21005.644} C_VEL
LIN {X 0,Y 238.812,Z 294.437,A -85,B 0,C 180,E1 -21006.402,E2 -21006.402} C_VEL
LIN {X 0,Y 239.91,Z 280.139,A -85,B 0,C 180,E1 -21006.92,E2 -21006.92} C_VEL
LIN {X 0,Y 241.869,Z 243.061,A -85,B 0,C 180,E1 -21008.031,E2 -21008.031} C_VEL
LIN {X 0,Y 240.762,Z 235.332,A -85,B 0,C 180,E1 -21008.624,E2 -21008.624} C_VEL
LIN {X 0,Y 235.58,Z 223.327,A -85,B 0,C 180,E1 -21010.451,E2 -21010.451} C_VEL
LIN {X 0,Y 230.213,Z 212.66,A -85,B 0,C 180,E1 -21012.456,E2 -21012.456} C_VEL
LIN {X 0,Y 225.244,Z 203.904,A -85,B 0,C 180,E1 -21014.421,E2 -21014.421} C_VEL
LIN {X 0,Y 220.46,Z 196.091,A -85,B 0,C 180,E1 -21016.451,E2 -21016.451} C_VEL
LIN {X 0,Y 216.788,Z 190.459,A -85,B 0,C 180,E1 -21018.146,E2 -21018.146} C_VEL
LIN {X 0,Y 213.64,Z 185.744,A -85,B 0,C 180,E1 -21019.712,E2 -21019.712} C_VEL
LIN {X 0,Y 209.188,Z 179.719,A -85,B 0,C 180,E1 -21022.092,E2 -21022.092} C_VEL
LIN {X 0,Y 208.668,Z 178.59,A -85,B 0,C 180,E1 -21022.495,E2 -21022.495} C_VEL
LIN {X 0,Y 207.31,Z 174.763,A -85,B 0,C 180,E1 -21025.987,E2 -21025.987} C_VEL
LIN {X 0,Y 206.711,Z 172.727,A -85,B 0,C 180,E1 -21028.209,E2 -21028.209} C_VEL
LIN {X 0,Y 206.71,Z 172.725,A -85,B 0,C 180,E1 -21032.127,E2 -21032.127} C_VEL
LIN {X 0,Y 206.732,Z 172.72,A -85,B 0,C 180,E1 -21036.618,E2 -21036.618} C_VEL
LIN {X 0,Y 206.804,Z 172.708,A -85,B 0,C 180,E1 -21042.189,E2 -21042.189} C_VEL
LIN {X 0,Y 206.857,Z 172.703,A -85,B 0,C 180,E1 -21046.241,E2 -21046.241} C_VEL
LIN {X 0,Y 207.075,Z 172.683,A -85,B 0,C 180,E1 -21050.229,E2 -21050.229} C_VEL
LIN {X 0,Y 207.04,Z 172.694,A -85,B 0,C 180,E1 -21054.154,E2 -21054.154} C_VEL
LIN {X 0,Y 207.347,Z 172.645,A -85,B 0,C 180,E1 -21058.057,E2 -21058.057} C_VEL
LIN {X 0,Y 207.484,Z 172.63,A -85,B 0,C 180,E1 -21059.999,E2 -21059.999} C_VEL
LIN {X 0,Y 207.377,Z 172.636,A -85,B 0,C 180,E1 -21061.941,E2 -21061.941} C_VEL
LIN {X 0,Y 207.131,Z 172.681,A -85,B 0,C 180,E1 -21067.799,E2 -21067.799} C_VEL
LIN {X 0,Y 206.922,Z 172.703,A -85,B 0,C 180,E1 -21071.757,E2 -21071.757} C_VEL
LIN {X 0,Y 206.902,Z 172.807,A -85,B 0,C 180,E1 -21076.844,E2 -21076.844} C_VEL
LIN {X 0,Y 207.687,Z 175.198,A -85,B 0,C 180,E1 -21077.412,E2 -21077.412} C_VEL
LIN {X 0,Y 209.517,Z 177.452,A -85,B 0,C 180,E1 -21078.454,E2 -21078.454} C_VEL
LIN {X 0,Y 211.098,Z 178.512,A -85,B 0,C 180,E1 -21079.256,E2 -21079.256} C_VEL
LIN {X 0,Y 212.829,Z 181.588,A -85,B 0,C 180,E1 -21080.223,E2 -21080.223} C_VEL
LIN {X 0,Y 215.346,Z 184.097,A -85,B 0,C 180,E1 -21081.437,E2 -21081.437} C_VEL
LIN {X 0,Y 217.54,Z 187.305,A -85,B 0,C 180,E1 -21082.503,E2 -21082.503} C_VEL
LIN {X 0,Y 219.201,Z 189.259,A -85,B 0,C 180,E1 -21083.25,E2 -21083.25} C_VEL
LIN {X 0,Y 223.008,Z 194.532,A -85,B 0,C 180,E1 -21084.895,E2 -21084.895} C_VEL
LIN {X 0,Y 227.754,Z 201.142,A -85,B 0,C 180,E1 -21086.778,E2 -21086.778} C_VEL
LIN {X 0,Y 232.934,Z 209.739,A -85,B 0,C 180,E1 -21088.734,E2 -21088.734} C_VEL
LIN {X 0,Y 238.361,Z 219.931,A -85,B 0,C 180,E1 -21090.663,E2 -21090.663} C_VEL
LIN {X 0,Y 242.754,Z 229.217,A -85,B 0,C 180,E1 -21092.139,E2 -21092.139} C_VEL
LIN {X 0,Y 239.817,Z 277.731,A -85,B 0,C 180,E1 -21093.584,E2 -21093.584} C_VEL
LIN {X 0,Y 238.135,Z 291.089,A -85,B 0,C 180,E1 -21094.274,E2 -21094.274} C_VEL
LIN {X 0,Y 236.13,Z 303.257,A -85,B 0,C 180,E1 -21095.251,E2 -21095.251} C_VEL
LIN {X 0,Y 233.203,Z 315.639,A -85,B 0,C 180,E1 -21096.576,E2 -21096.576} C_VEL
LIN {X 0,Y 230.096,Z 326.639,A -85,B 0,C 180,E1 -21098.14,E2 -21098.14} C_VEL
LIN {X 0,Y 226.779,Z 336.467,A -85,B 0,C 180,E1 -21099.906,E2 -21099.906} C_VEL
LIN {X 0,Y 222.906,Z 346.376,A -85,B 0,C 180,E1 -21102.189,E2 -21102.189} C_VEL
LIN {X 0,Y 219.308,Z 354.54,A -85,B 0,C 180,E1 -21104.584,E2 -21104.584} C_VEL
LIN {X 0,Y 215.628,Z 362.139,A -85,B 0,C 180,E1 -21107.444,E2 -21107.444} C_VEL
LIN {X 0,Y 212.875,Z 367.429,A -85,B 0,C 180,E1 -21110.028,E2 -21110.028} C_VEL
LIN {X 0,Y 209.919,Z 372.69,A -85,B 0,C 180,E1 -21113.465,E2 -21113.465} C_VEL
LIN {X 0,Y 207.486,Z 376.613,A -85,B 0,C 180,E1 -21117.183,E2 -21117.183} C_VEL
LIN {X 0,Y 206.434,Z 378.077,A -85,B 0,C 180,E1 -21119.292,E2 -21119.292} C_VEL
LIN {X 0,Y 205.135,Z 379.513,A -85,B 0,C 180,E1 -21122.967,E2 -21122.967} C_VEL
LIN {X 0,Y 204.501,Z 379.697,A -85,B 0,C 180,E1 -21125.645,E2 -21125.645} C_VEL
LIN {X 0,Y 204.222,Z 379.179,A -85,B 0,C 180,E1 -21128.302,E2 -21128.302} C_VEL
LIN {X 0,Y 204.144,Z 377.252,A -85,B 0,C 180,E1 -21131.951,E2 -21131.951} C_VEL
LIN {X 0,Y 204.39,Z 375.266,A -85,B 0,C 180,E1 -21134.316,E2 -21134.316} C_VEL
LIN {X 0,Y 204.855,Z 372.072,A -85,B 0,C 180,E1 -21137.115,E2 -21137.115} C_VEL
LIN {X 0,Y 205.594,Z 367.493,A -85,B 0,C 180,E1 -21140.159,E2 -21140.159} C_VEL
LIN {X 0,Y 206.66,Z 361.665,A -85,B 0,C 180,E1 -21143.164,E2 -21143.164} C_VEL
LIN {X 0,Y 208.12,Z 354.324,A -85,B 0,C 180,E1 -21146.128,E2 -21146.128} C_VEL
LIN {X 0,Y 209.991,Z 345.172,A -85,B 0,C 180,E1 -21149.041,E2 -21149.041} C_VEL
LIN {X 0,Y 211.982,Z 335.442,A -85,B 0,C 180,E1 -21151.487,E2 -21151.487} C_VEL
LIN {X 0,Y 213.832,Z 325.196,A -85,B 0,C 180,E1 -21153.533,E2 -21153.533} C_VEL
LIN {X 0,Y 215.516,Z 315.086,A -85,B 0,C 180,E1 -21155.145,E2 -21155.145} C_VEL
LIN {X 0,Y 217.063,Z 303.336,A -85,B 0,C 180,E1 -21156.624,E2 -21156.624} C_VEL
LIN {X 0,Y 218.448,Z 290.528,A -85,B 0,C 180,E1 -21157.801,E2 -21157.801} C_VEL
LIN {X 0,Y 219.385,Z 278.086,A -85,B 0,C 180,E1 -21158.579,E2 -21158.579} C_VEL
LIN {X 0,Y 220.318,Z 256.918,A -85,B 0,C 180,E1 -21159.329,E2 -21159.329} C_VEL
LIN {X 0,Y 222.124,Z 209.801,A -85,B 0,C 180,E1 -21160.82,E2 -21160.82} C_VEL
LIN {X 0,Y 216.28,Z 192.708,A -85,B 0,C 180,E1 -21162.174,E2 -21162.174} C_VEL
LIN {X 0,Y 208.088,Z 175.98,A -85,B 0,C 180,E1 -21163.925,E2 -21163.925} C_VEL
LIN {X 0,Y 206.917,Z 173.273,A -85,B 0,C 180,E1 -21164.201,E2 -21164.201} C_VEL
LIN {X 0,Y 206.814,Z 172.727,A -85,B 0,C 180,E1 -21164.263,E2 -21164.263} C_VEL
LIN {X 0,Y 206.805,Z 172.726,A -85,B 0,C 180,E1 -21167.913,E2 -21167.913} C_VEL
LIN {X 0,Y 206.706,Z 172.708,A -85,B 0,C 180,E1 -21173.368,E2 -21173.368} C_VEL
LIN {X 0,Y 206.675,Z 172.723,A -85,B 0,C 180,E1 -21178.43,E2 -21178.43} C_VEL
LIN {X 0,Y 206.692,Z 172.739,A -85,B 0,C 180,E1 -21182.96,E2 -21182.96} C_VEL
LIN {X 0,Y 206.666,Z 172.731,A -85,B 0,C 180,E1 -21187.744,E2 -21187.744} C_VEL
LIN {X 0,Y 206.629,Z 172.745,A -85,B 0,C 180,E1 -21191.56,E2 -21191.56} C_VEL
LIN {X 0,Y 206.628,Z 172.724,A -85,B 0,C 180,E1 -21195.584,E2 -21195.584} C_VEL
LIN {X 0,Y 206.646,Z 172.734,A -85,B 0,C 180,E1 -21199.747,E2 -21199.747} C_VEL
LIN {X 0,Y 206.699,Z 172.734,A -85,B 0,C 180,E1 -21204.69,E2 -21204.69} C_VEL
LIN {X 0,Y 206.694,Z 172.704,A -85,B 0,C 180,E1 -21209.336,E2 -21209.336} C_VEL
LIN {X 0,Y 206.684,Z 172.723,A -85,B 0,C 180,E1 -21213.767,E2 -21213.767} C_VEL
LIN {X 0,Y 206.708,Z 172.736,A -85,B 0,C 180,E1 -21218.039,E2 -21218.039} C_VEL
LIN {X 0,Y 206.804,Z 172.716,A -85,B 0,C 180,E1 -21222.192,E2 -21222.192} C_VEL
LIN {X 0,Y 206.849,Z 172.721,A -85,B 0,C 180,E1 -21226.242,E2 -21226.242} C_VEL
LIN {X 0,Y 207.076,Z 172.682,A -85,B 0,C 180,E1 -21230.231,E2 -21230.231} C_VEL
LIN {X 0,Y 207.038,Z 172.697,A -85,B 0,C 180,E1 -21234.156,E2 -21234.156} C_VEL
LIN {X 0,Y 207.345,Z 172.652,A -85,B 0,C 180,E1 -21238.059,E2 -21238.059} C_VEL
LIN {X 0,Y 207.483,Z 172.632,A -85,B 0,C 180,E1 -21240.001,E2 -21240.001} C_VEL
LIN {X 0,Y 207.347,Z 172.655,A -85,B 0,C 180,E1 -21241.943,E2 -21241.943} C_VEL
LIN {X 0,Y 207.129,Z 172.676,A -85,B 0,C 180,E1 -21247.801,E2 -21247.801} C_VEL
LIN {X 0,Y 206.913,Z 172.713,A -85,B 0,C 180,E1 -21251.76,E2 -21251.76} C_VEL
LIN {X 0,Y 206.806,Z 172.715,A -85,B 0,C 180,E1 -21255.777,E2 -21255.777} C_VEL
LIN {X 0,Y 206.717,Z 172.735,A -85,B 0,C 180,E1 -21259.877,E2 -21259.877} C_VEL
LIN {X 0,Y 206.739,Z 172.731,A -85,B 0,C 180,E1 -21264.076,E2 -21264.076} C_VEL
LIN {X 0,Y 206.693,Z 172.737,A -85,B 0,C 180,E1 -21268.428,E2 -21268.428} C_VEL
LIN {X 0,Y 206.699,Z 172.739,A -85,B 0,C 180,E1 -21272.959,E2 -21272.959} C_VEL
LIN {X 0,Y 206.672,Z 172.741,A -85,B 0,C 180,E1 -21277.743,E2 -21277.743} C_VEL
LIN {X 0,Y 206.635,Z 172.749,A -85,B 0,C 180,E1 -21281.559,E2 -21281.559} C_VEL
LIN {X 0,Y 206.634,Z 172.749,A -85,B 0,C 180,E1 -21285.583,E2 -21285.583} C_VEL
LIN {X 0,Y 206.654,Z 172.744,A -85,B 0,C 180,E1 -21289.746,E2 -21289.746} C_VEL
LIN {X 0,Y 206.687,Z 172.763,A -85,B 0,C 180,E1 -21291.741,E2 -21291.741} C_VEL
LIN {X 0,Y 206.889,Z 173.617,A -85,B 0,C 180,E1 -21292.146,E2 -21292.146} C_VEL
LIN {X 0,Y 206.823,Z 176.034,A -85,B 0,C 180,E1 -21293.06,E2 -21293.06} C_VEL
LIN {X 0,Y 205.997,Z 178.96,A -85,B 0,C 180,E1 -21293.846,E2 -21293.846} C_VEL
LIN {X 0,Y 204.514,Z 184.517,A -85,B 0,C 180,E1 -21294.915,E2 -21294.915} C_VEL
LIN {X 0,Y 204.535,Z 188.746,A -85,B 0,C 180,E1 -21295.508,E2 -21295.508} C_VEL
LIN {X 0,Y 205.093,Z 190.538,A -85,B 0,C 180,E1 -21295.71,E2 -21295.71} C_VEL
LIN {X 0,Y 211.404,Z 207.932,A -85,B 0,C 180,E1 -21297.252,E2 -21297.252} C_VEL
LIN {X 0,Y 214.77,Z 237.164,A -85,B 0,C 180,E1 -21298.783,E2 -21298.783} C_VEL
LIN {X 0,Y 212.716,Z 290.208,A -85,B 0,C 180,E1 -21300.563,E2 -21300.563} C_VEL
LIN {X 0,Y 211.607,Z 303.441,A -85,B 0,C 180,E1 -21301.346,E2 -21301.346} C_VEL
LIN {X 0,Y 210.01,Z 316.183,A -85,B 0,C 180,E1 -21302.468,E2 -21302.468} C_VEL
LIN {X 0,Y 208.144,Z 328.344,A -85,B 0,C 180,E1 -21303.963,E2 -21303.963} C_VEL
LIN {X 0,Y 206.317,Z 338.632,A -85,B 0,C 180,E1 -21305.604,E2 -21305.604} C_VEL
LIN {X 0,Y 204.387,Z 348.21,A -85,B 0,C 180,E1 -21307.508,E2 -21307.508} C_VEL
LIN {X 0,Y 202.967,Z 355.318,A -85,B 0,C 180,E1 -21309.216,E2 -21309.216} C_VEL
LIN {X 0,Y 201.291,Z 363.777,A -85,B 0,C 180,E1 -21311.685,E2 -21311.685} C_VEL
LIN {X 0,Y 199.624,Z 372.04,A -85,B 0,C 180,E1 -21314.689,E2 -21314.689} C_VEL
LIN {X 0,Y 198.42,Z 378.668,A -85,B 0,C 180,E1 -21317.73,E2 -21317.73} C_VEL
LIN {X 0,Y 197.751,Z 383.927,A -85,B 0,C 180,E1 -21320.797,E2 -21320.797} C_VEL
LIN {X 0,Y 197.409,Z 387.978,A -85,B 0,C 180,E1 -21323.868,E2 -21323.868} C_VEL
LIN {X 0,Y 197.328,Z 390.053,A -85,B 0,C 180,E1 -21325.915,E2 -21325.915} C_VEL
LIN {X 0,Y 197.4,Z 391.693,A -85,B 0,C 180,E1 -21327.959,E2 -21327.959} C_VEL
LIN {X 0,Y 197.513,Z 392.918,A -85,B 0,C 180,E1 -21330,E2 -21330} C_VEL
LIN {X 0,Y 197.369,Z 393.71,A -85,B 0,C 180,E1 -21332.04,E2 -21332.04} C_VEL
LIN {X 0,Y 197.337,Z 394.046,A -85,B 0,C 180,E1 -21336.133,E2 -21336.133} C_VEL
LIN {X 0,Y 197.99,Z 392.864,A -85,B 0,C 180,E1 -21340.223,E2 -21340.223} C_VEL
LIN {X 0,Y 198.641,Z 391.661,A -85,B 0,C 180,E1 -21342.256,E2 -21342.256} C_VEL
LIN {X 0,Y 200.614,Z 388.044,A -85,B 0,C 180,E1 -21346.275,E2 -21346.275} C_VEL
LIN {X 0,Y 202.899,Z 384.181,A -85,B 0,C 180,E1 -21349.212,E2 -21349.212} C_VEL
LIN {X 0,Y 205.543,Z 379.229,A -85,B 0,C 180,E1 -21352.093,E2 -21352.093} C_VEL
LIN {X 0,Y 208.633,Z 373.045,A -85,B 0,C 180,E1 -21354.902,E2 -21354.902} C_VEL
LIN {X 0,Y 212.391,Z 365.383,A -85,B 0,C 180,E1 -21357.597,E2 -21357.597} C_VEL
LIN {X 0,Y 216.729,Z 355.802,A -85,B 0,C 180,E1 -21360.174,E2 -21360.174} C_VEL
LIN {X 0,Y 220.254,Z 347.023,A -85,B 0,C 180,E1 -21362.038,E2 -21362.038} C_VEL
LIN {X 0,Y 223.596,Z 337.602,A -85,B 0,C 180,E1 -21363.641,E2 -21363.641} C_VEL
LIN {X 0,Y 227.196,Z 325.934,A -85,B 0,C 180,E1 -21365.179,E2 -21365.179} C_VEL
LIN {X 0,Y 230.3,Z 313.494,A -85,B 0,C 180,E1 -21366.382,E2 -21366.382} C_VEL
LIN {X 0,Y 232.793,Z 300.58,A -85,B 0,C 180,E1 -21367.265,E2 -21367.265} C_VEL
LIN {X 0,Y 234.273,Z 288.311,A -85,B 0,C 180,E1 -21367.845,E2 -21367.845} C_VEL
LIN {X 0,Y 236.835,Z 244.742,A -85,B 0,C 180,E1 -21369.171,E2 -21369.171} C_VEL
LIN {X 0,Y 235.931,Z 238.361,A -85,B 0,C 180,E1 -21369.682,E2 -21369.682} C_VEL
LIN {X 0,Y 231.273,Z 227.382,A -85,B 0,C 180,E1 -21371.439,E2 -21371.439} C_VEL
LIN {X 0,Y 225.758,Z 216.09,A -85,B 0,C 180,E1 -21373.629,E2 -21373.629} C_VEL
LIN {X 0,Y 219.742,Z 205.639,A -85,B 0,C 180,E1 -21376.172,E2 -21376.172} C_VEL
LIN {X 0,Y 216.692,Z 200.717,A -85,B 0,C 180,E1 -21377.573,E2 -21377.573} C_VEL
LIN {X 0,Y 213.634,Z 195.893,A -85,B 0,C 180,E1 -21379.076,E2 -21379.076} C_VEL
LIN {X 0,Y 209.992,Z 190.417,A -85,B 0,C 180,E1 -21380.993,E2 -21380.993} C_VEL
LIN {X 0,Y 206.412,Z 185.228,A -85,B 0,C 180,E1 -21383.045,E2 -21383.045} C_VEL
LIN {X 0,Y 201.828,Z 179.33,A -85,B 0,C 180,E1 -21385.99,E2 -21385.99} C_VEL
LIN {X 0,Y 201.11,Z 178.016,A -85,B 0,C 180,E1 -21386.57,E2 -21386.57} C_VEL
LIN {X 0,Y 200.609,Z 176.346,A -85,B 0,C 180,E1 -21388.297,E2 -21388.297} C_VEL
LIN {X 0,Y 199.666,Z 173.607,A -85,B 0,C 180,E1 -21391.639,E2 -21391.639} C_VEL
LIN {X 0,Y 199.674,Z 173.596,A -85,B 0,C 180,E1 -21397.22,E2 -21397.22} C_VEL
LIN {X 0,Y 199.747,Z 173.587,A -85,B 0,C 180,E1 -21401.802,E2 -21401.802} C_VEL
LIN {X 0,Y 199.796,Z 173.586,A -85,B 0,C 180,E1 -21405.744,E2 -21405.744} C_VEL
LIN {X 0,Y 200.024,Z 173.566,A -85,B 0,C 180,E1 -21409.881,E2 -21409.881} C_VEL
LIN {X 0,Y 200.003,Z 173.568,A -85,B 0,C 180,E1 -21413.948,E2 -21413.948} C_VEL
LIN {X 0,Y 200.289,Z 173.523,A -85,B 0,C 180,E1 -21417.988,E2 -21417.988} C_VEL
LIN {X 0,Y 200.451,Z 173.505,A -85,B 0,C 180,E1 -21419.999,E2 -21419.999} C_VEL
LIN {X 0,Y 200.317,Z 173.516,A -85,B 0,C 180,E1 -21422.01,E2 -21422.01} C_VEL
LIN {X 0,Y 200.078,Z 173.562,A -85,B 0,C 180,E1 -21428.076,E2 -21428.076} C_VEL
LIN {X 0,Y 199.872,Z 173.585,A -85,B 0,C 180,E1 -21432.178,E2 -21432.178} C_VEL
LIN {X 0,Y 199.829,Z 173.595,A -85,B 0,C 180,E1 -21432.826,E2 -21432.826} C_VEL
LIN {X 0,Y 200.553,Z 175.875,A -85,B 0,C 180,E1 -21433.488,E2 -21433.488} C_VEL
LIN {X 0,Y 202.273,Z 178.143,A -85,B 0,C 180,E1 -21434.718,E2 -21434.718} C_VEL
LIN {X 0,Y 204.481,Z 179.597,A -85,B 0,C 180,E1 -21436.079,E2 -21436.079} C_VEL
LIN {X 0,Y 206.284,Z 182.783,A -85,B 0,C 180,E1 -21437.264,E2 -21437.264} C_VEL
LIN {X 0,Y 208.736,Z 185.165,A -85,B 0,C 180,E1 -21438.621,E2 -21438.621} C_VEL
LIN {X 0,Y 211.14,Z 188.647,A -85,B 0,C 180,E1 -21439.948,E2 -21439.948} C_VEL
LIN {X 0,Y 212.721,Z 190.329,A -85,B 0,C 180,E1 -21440.739,E2 -21440.739} C_VEL
LIN {X 0,Y 215.57,Z 194.084,A -85,B 0,C 180,E1 -21442.139,E2 -21442.139} C_VEL
LIN {X 0,Y 219.788,Z 200.027,A -85,B 0,C 180,E1 -21444.083,E2 -21444.083} C_VEL
LIN {X 0,Y 224.525,Z 206.818,A -85,B 0,C 180,E1 -21446.05,E2 -21446.05} C_VEL
LIN {X 0,Y 229.171,Z 214.695,A -85,B 0,C 180,E1 -21447.886,E2 -21447.886} C_VEL
LIN {X 0,Y 234.349,Z 224.679,A -85,B 0,C 180,E1 -21449.828,E2 -21449.828} C_VEL
LIN {X 0,Y 237.636,Z 232.002,A -85,B 0,C 180,E1 -21451.016,E2 -21451.016} C_VEL
LIN {X 0,Y 234.761,Z 277.63,A -85,B 0,C 180,E1 -21452.388,E2 -21452.388} C_VEL
LIN {X 0,Y 232.992,Z 291.182,A -85,B 0,C 180,E1 -21453.085,E2 -21453.085} C_VEL
LIN {X 0,Y 230.797,Z 303.883,A -85,B 0,C 180,E1 -21454.118,E2 -21454.118} C_VEL
LIN {X 0,Y 227.669,Z 316.477,A -85,B 0,C 180,E1 -21455.494,E2 -21455.494} C_VEL
LIN {X 0,Y 224.507,Z 327.116,A -85,B 0,C 180,E1 -21457.036,E2 -21457.036} C_VEL
LIN {X 0,Y 221.055,Z 336.93,A -85,B 0,C 180,E1 -21458.837,E2 -21458.837} C_VEL
LIN {X 0,Y 217.009,Z 346.774,A -85,B 0,C 180,E1 -21461.152,E2 -21461.152} C_VEL
LIN {X 0,Y 213.319,Z 354.769,A -85,B 0,C 180,E1 -21463.547,E2 -21463.547} C_VEL
LIN {X 0,Y 209.356,Z 362.486,A -85,B 0,C 180,E1 -21466.514,E2 -21466.514} C_VEL
LIN {X 0,Y 206.008,Z 368.483,A -85,B 0,C 180,E1 -21469.595,E2 -21469.595} C_VEL
LIN {X 0,Y 203.314,Z 372.96,A -85,B 0,C 180,E1 -21472.658,E2 -21472.658} C_VEL
LIN {X 0,Y 201.013,Z 376.441,A -85,B 0,C 180,E1 -21475.985,E2 -21475.985} C_VEL
LIN {X 0,Y 199.821,Z 378.059,A -85,B 0,C 180,E1 -21478.159,E2 -21478.159} C_VEL
LIN {X 0,Y 198.854,Z 379.149,A -85,B 0,C 180,E1 -21480.344,E2 -21480.344} C_VEL
LIN {X 0,Y 198.145,Z 379.792,A -85,B 0,C 180,E1 -21482.542,E2 -21482.542} C_VEL
LIN {X 0,Y 197.569,Z 380.004,A -85,B 0,C 180,E1 -21484.731,E2 -21484.731} C_VEL
LIN {X 0,Y 197.15,Z 379.462,A -85,B 0,C 180,E1 -21487.946,E2 -21487.946} C_VEL
LIN {X 0,Y 197.032,Z 377.877,A -85,B 0,C 180,E1 -21491.275,E2 -21491.275} C_VEL
LIN {X 0,Y 197.261,Z 375.62,A -85,B 0,C 180,E1 -21494.14,E2 -21494.14} C_VEL
LIN {X 0,Y 197.867,Z 371.643,A -85,B 0,C 180,E1 -21497.695,E2 -21497.695} C_VEL
LIN {X 0,Y 198.679,Z 366.861,A -85,B 0,C 180,E1 -21500.83,E2 -21500.83} C_VEL
LIN {X 0,Y 199.875,Z 360.735,A -85,B 0,C 180,E1 -21503.945,E2 -21503.945} C_VEL
LIN {X 0,Y 201.434,Z 353.128,A -85,B 0,C 180,E1 -21507,E2 -21507} C_VEL
LIN {X 0,Y 203.116,Z 345.348,A -85,B 0,C 180,E1 -21509.505,E2 -21509.505} C_VEL
LIN {X 0,Y 204.773,Z 337.359,A -85,B 0,C 180,E1 -21511.613,E2 -21511.613} C_VEL
LIN {X 0,Y 206.82,Z 326.662,A -85,B 0,C 180,E1 -21513.897,E2 -21513.897} C_VEL
LIN {X 0,Y 208.861,Z 315.185,A -85,B 0,C 180,E1 -21515.794,E2 -21515.794} C_VEL
LIN {X 0,Y 210.458,Z 303.404,A -85,B 0,C 180,E1 -21517.315,E2 -21517.315} C_VEL
LIN {X 0,Y 211.899,Z 290.497,A -85,B 0,C 180,E1 -21518.524,E2 -21518.524} C_VEL
LIN {X 0,Y 212.875,Z 277.919,A -85,B 0,C 180,E1 -21519.322,E2 -21519.322} C_VEL
LIN {X 0,Y 213.971,Z 252.626,A -85,B 0,C 180,E1 -21520.223,E2 -21520.223} C_VEL
LIN {X 0,Y 215.611,Z 211.193,A -85,B 0,C 180,E1 -21521.57,E2 -21521.57} C_VEL
LIN {X 0,Y 210.171,Z 195.307,A -85,B 0,C 180,E1 -21522.88,E2 -21522.88} C_VEL
LIN {X 0,Y 202.608,Z 179.854,A -85,B 0,C 180,E1 -21524.57,E2 -21524.57} C_VEL
LIN {X 0,Y 199.929,Z 174.42,A -85,B 0,C 180,E1 -21525.203,E2 -21525.203} C_VEL
LIN {X 0,Y 199.767,Z 173.604,A -85,B 0,C 180,E1 -21525.301,E2 -21525.301} C_VEL
LIN {X 0,Y 199.72,Z 173.607,A -85,B 0,C 180,E1 -21528.464,E2 -21528.464} C_VEL
LIN {X 0,Y 199.67,Z 173.576,A -85,B 0,C 180,E1 -21533.776,E2 -21533.776} C_VEL
LIN {X 0,Y 199.652,Z 173.595,A -85,B 0,C 180,E1 -21538.357,E2 -21538.357} C_VEL
LIN {X 0,Y 199.663,Z 173.614,A -85,B 0,C 180,E1 -21542.353,E2 -21542.353} C_VEL
LIN {X 0,Y 199.615,Z 173.601,A -85,B 0,C 180,E1 -21546.766,E2 -21546.766} C_VEL
LIN {X 0,Y 199.592,Z 173.62,A -85,B 0,C 180,E1 -21549.333,E2 -21549.333} C_VEL
LIN {X 0,Y 199.564,Z 173.624,A -85,B 0,C 180,E1 -21552.309,E2 -21552.309} C_VEL
LIN {X 0,Y 199.574,Z 173.603,A -85,B 0,C 180,E1 -21555.229,E2 -21555.229} C_VEL
LIN {X 0,Y 199.569,Z 173.602,A -85,B 0,C 180,E1 -21558.004,E2 -21558.004} C_VEL
LIN {X 0,Y 199.596,Z 173.616,A -85,B 0,C 180,E1 -21560.774,E2 -21560.774} C_VEL
LIN {X 0,Y 199.61,Z 173.613,A -85,B 0,C 180,E1 -21565.715,E2 -21565.715} C_VEL
LIN {X 0,Y 199.685,Z 173.584,A -85,B 0,C 180,E1 -21568.136,E2 -21568.136} C_VEL
LIN {X 0,Y 199.634,Z 173.59,A -85,B 0,C 180,E1 -21572.765,E2 -21572.765} C_VEL
LIN {X 0,Y 199.669,Z 173.612,A -85,B 0,C 180,E1 -21577.222,E2 -21577.222} C_VEL
LIN {X 0,Y 199.747,Z 173.596,A -85,B 0,C 180,E1 -21581.804,E2 -21581.804} C_VEL
LIN {X 0,Y 199.769,Z 173.6,A -85,B 0,C 180,E1 -21585.745,E2 -21585.745} C_VEL
LIN {X 0,Y 200.025,Z 173.562,A -85,B 0,C 180,E1 -21589.883,E2 -21589.883} C_VEL
LIN {X 0,Y 200.001,Z 173.571,A -85,B 0,C 180,E1 -21593.95,E2 -21593.95} C_VEL
LIN {X 0,Y 200.287,Z 173.532,A -85,B 0,C 180,E1 -21597.99,E2 -21597.99} C_VEL
LIN {X 0,Y 200.45,Z 173.507,A -85,B 0,C 180,E1 -21600.001,E2 -21600.001} C_VEL
LIN {X 0,Y 199.992,Z 173.575,A -85,B 0,C 180,E1 -21604.031,E2 -21604.031} C_VEL
LIN {X 0,Y 200.077,Z 173.553,A -85,B 0,C 180,E1 -21608.078,E2 -21608.078} C_VEL
LIN {X 0,Y 199.861,Z 173.59,A -85,B 0,C 180,E1 -21612.181,E2 -21612.181} C_VEL
LIN {X 0,Y 199.746,Z 173.594,A -85,B 0,C 180,E1 -21616.35,E2 -21616.35} C_VEL
LIN {X 0,Y 199.65,Z 173.615,A -85,B 0,C 180,E1 -21620.612,E2 -21620.612} C_VEL
LIN {X 0,Y 199.653,Z 173.615,A -85,B 0,C 180,E1 -21624.988,E2 -21624.988} C_VEL
LIN {X 0,Y 199.613,Z 173.62,A -85,B 0,C 180,E1 -21629.533,E2 -21629.533} C_VEL
LIN {X 0,Y 199.67,Z 173.613,A -85,B 0,C 180,E1 -21632.353,E2 -21632.353} C_VEL
LIN {X 0,Y 199.621,Z 173.622,A -85,B 0,C 180,E1 -21636.765,E2 -21636.765} C_VEL
LIN {X 0,Y 199.598,Z 173.625,A -85,B 0,C 180,E1 -21639.332,E2 -21639.332} C_VEL
LIN {X 0,Y 199.57,Z 173.63,A -85,B 0,C 180,E1 -21642.308,E2 -21642.308} C_VEL
LIN {X 0,Y 199.58,Z 173.629,A -85,B 0,C 180,E1 -21645.228,E2 -21645.228} C_VEL
LIN {X 0,Y 199.576,Z 173.626,A -85,B 0,C 180,E1 -21648.003,E2 -21648.003} C_VEL
LIN {X 0,Y 199.646,Z 173.739,A -85,B 0,C 180,E1 -21651.076,E2 -21651.076} C_VEL
LIN {X 0,Y 201.52,Z 181.694,A -85,B 0,C 180,E1 -21654.825,E2 -21654.825} C_VEL
LIN {X 0,Y 205.093,Z 190.538,A -85,B 0,C 180,E1 -21655.71,E2 -21655.71} C_VEL
LIN {X 0,Y 206.254,Z 194.131,A -85,B 0,C 180,E1 -21656.018,E2 -21656.018} C_VEL
LIN {X 0,Y 206.933,Z 199.913,A -85,B 0,C 180,E1 -21656.341,E2 -21656.341} C_VEL
LIN {X 0,Y 206.206,Z 218.001,A -85,B 0,C 180,E1 -21656.951,E2 -21656.951} C_VEL
LIN {X 0,Y 206.515,Z 221.991,A -85,B 0,C 180,E1 -21657.15,E2 -21657.15} C_VEL
LIN {X 0,Y 208.296,Z 238.692,A -85,B 0,C 180,E1 -21658.032,E2 -21658.032} C_VEL
LIN {X 0,Y 206.18,Z 290.333,A -85,B 0,C 180,E1 -21659.815,E2 -21659.815} C_VEL
LIN {X 0,Y 204.93,Z 304.196,A -85,B 0,C 180,E1 -21660.674,E2 -21660.674} C_VEL
LIN {X 0,Y 203.218,Z 317.18,A -85,B 0,C 180,E1 -21661.887,E2 -21661.887} C_VEL
LIN {X 0,Y 201.453,Z 328.23,A -85,B 0,C 180,E1 -21663.309,E2 -21663.309} C_VEL
LIN {X 0,Y 199.554,Z 338.494,A -85,B 0,C 180,E1 -21664.999,E2 -21664.999} C_VEL
LIN {X 0,Y 197.571,Z 348.057,A -85,B 0,C 180,E1 -21666.964,E2 -21666.964} C_VEL
LIN {X 0,Y 195.864,Z 356.031,A -85,B 0,C 180,E1 -21668.972,E2 -21668.972} C_VEL
LIN {X 0,Y 194.151,Z 364.348,A -85,B 0,C 180,E1 -21671.534,E2 -21671.534} C_VEL
LIN {X 0,Y 192.465,Z 372.471,A -85,B 0,C 180,E1 -21674.648,E2 -21674.648} C_VEL
LIN {X 0,Y 191.428,Z 377.953,A -85,B 0,C 180,E1 -21677.274,E2 -21677.274} C_VEL
LIN {X 0,Y 190.708,Z 383.309,A -85,B 0,C 180,E1 -21680.454,E2 -21680.454} C_VEL
LIN {X 0,Y 190.349,Z 387.446,A -85,B 0,C 180,E1 -21683.64,E2 -21683.64} C_VEL
LIN {X 0,Y 190.244,Z 389.716,A -85,B 0,C 180,E1 -21685.908,E2 -21685.908} C_VEL
LIN {X 0,Y 190.3,Z 391.27,A -85,B 0,C 180,E1 -21687.883,E2 -21687.883} C_VEL
LIN {X 0,Y 190.429,Z 392.532,A -85,B 0,C 180,E1 -21690,E2 -21690} C_VEL
LIN {X 0,Y 190.164,Z 393.724,A -85,B 0,C 180,E1 -21693.74,E2 -21693.74} C_VEL
LIN {X 0,Y 190.275,Z 393.803,A -85,B 0,C 180,E1 -21696.362,E2 -21696.362} C_VEL
LIN {X 0,Y 190.991,Z 392.702,A -85,B 0,C 180,E1 -21700.602,E2 -21700.602} C_VEL
LIN {X 0,Y 191.681,Z 391.572,A -85,B 0,C 180,E1 -21702.708,E2 -21702.708} C_VEL
LIN {X 0,Y 192.562,Z 390.008,A -85,B 0,C 180,E1 -21704.802,E2 -21704.802} C_VEL
LIN {X 0,Y 194.525,Z 386.908,A -85,B 0,C 180,E1 -21707.884,E2 -21707.884} C_VEL
LIN {X 0,Y 197.026,Z 382.785,A -85,B 0,C 180,E1 -21710.898,E2 -21710.898} C_VEL
LIN {X 0,Y 200.319,Z 376.814,A -85,B 0,C 180,E1 -21714.189,E2 -21714.189} C_VEL
LIN {X 0,Y 204.125,Z 369.752,A -85,B 0,C 180,E1 -21717.142,E2 -21717.142} C_VEL
LIN {X 0,Y 208.359,Z 361.368,A -85,B 0,C 180,E1 -21719.836,E2 -21719.836} C_VEL
LIN {X 0,Y 212.268,Z 352.77,A -85,B 0,C 180,E1 -21721.988,E2 -21721.988} C_VEL
LIN {X 0,Y 216.386,Z 342.24,A -85,B 0,C 180,E1 -21724.074,E2 -21724.074} C_VEL
LIN {X 0,Y 220.076,Z 331.799,A -85,B 0,C 180,E1 -21725.648,E2 -21725.648} C_VEL
LIN {X 0,Y 223.462,Z 320.301,A -85,B 0,C 180,E1 -21726.977,E2 -21726.977} C_VEL
LIN {X 0,Y 226.44,Z 307.175,A -85,B 0,C 180,E1 -21728.087,E2 -21728.087} C_VEL
LIN {X 0,Y 228.59,Z 294.329,A -85,B 0,C 180,E1 -21728.827,E2 -21728.827} C_VEL
LIN {X 0,Y 229.879,Z 279.26,A -85,B 0,C 180,E1 -21729.383,E2 -21729.383} C_VEL
LIN {X 0,Y 231.869,Z 245.866,A -85,B 0,C 180,E1 -21730.403,E2 -21730.403} C_VEL
LIN {X 0,Y 231.283,Z 241.546,A -85,B 0,C 180,E1 -21730.765,E2 -21730.765} C_VEL
LIN {X 0,Y 226.701,Z 230.669,A -85,B 0,C 180,E1 -21732.603,E2 -21732.603} C_VEL
LIN {X 0,Y 221.922,Z 220.789,A -85,B 0,C 180,E1 -21734.608,E2 -21734.608} C_VEL
LIN {X 0,Y 216.414,Z 210.899,A -85,B 0,C 180,E1 -21737.078,E2 -21737.078} C_VEL
LIN {X 0,Y 213.392,Z 205.866,A -85,B 0,C 180,E1 -21738.556,E2 -21738.556} C_VEL
LIN {X 0,Y 210.577,Z 201.352,A -85,B 0,C 180,E1 -21740.015,E2 -21740.015} C_VEL
LIN {X 0,Y 207.431,Z 196.414,A -85,B 0,C 180,E1 -21741.761,E2 -21741.761} C_VEL
LIN {X 0,Y 203.223,Z 190.362,A -85,B 0,C 180,E1 -21744.31,E2 -21744.31} C_VEL
LIN {X 0,Y 199.566,Z 185.337,A -85,B 0,C 180,E1 -21746.847,E2 -21746.847} C_VEL
LIN {X 0,Y 198.335,Z 183.732,A -85,B 0,C 180,E1 -21747.772,E2 -21747.772} C_VEL
LIN {X 0,Y 194.361,Z 178.759,A -85,B 0,C 180,E1 -21751.096,E2 -21751.096} C_VEL
LIN {X 0,Y 193.569,Z 177.229,A -85,B 0,C 180,E1 -21751.982,E2 -21751.982} C_VEL
LIN {X 0,Y 192.667,Z 174.473,A -85,B 0,C 180,E1 -21756.342,E2 -21756.342} C_VEL
LIN {X 0,Y 192.696,Z 174.466,A -85,B 0,C 180,E1 -21761.491,E2 -21761.491} C_VEL
LIN {X 0,Y 192.722,Z 174.472,A -85,B 0,C 180,E1 -21765.209,E2 -21765.209} C_VEL
LIN {X 0,Y 192.947,Z 174.45,A -85,B 0,C 180,E1 -21769.566,E2 -21769.566} C_VEL
LIN {X 0,Y 192.967,Z 174.442,A -85,B 0,C 180,E1 -21773.726,E2 -21773.726} C_VEL
LIN {X 0,Y 193.233,Z 174.401,A -85,B 0,C 180,E1 -21777.915,E2 -21777.915} C_VEL
LIN {X 0,Y 193.417,Z 174.381,A -85,B 0,C 180,E1 -21779.999,E2 -21779.999} C_VEL
LIN {X 0,Y 192.962,Z 174.444,A -85,B 0,C 180,E1 -21784.176,E2 -21784.176} C_VEL
LIN {X 0,Y 193.066,Z 174.637,A -85,B 0,C 180,E1 -21787.91,E2 -21787.91} C_VEL
LIN {X 0,Y 193.791,Z 176.909,A -85,B 0,C 180,E1 -21788.799,E2 -21788.799} C_VEL
LIN {X 0,Y 195.704,Z 179.232,A -85,B 0,C 180,E1 -21790.525,E2 -21790.525} C_VEL
LIN {X 0,Y 197.705,Z 180.444,A -85,B 0,C 180,E1 -21792.053,E2 -21792.053} C_VEL
LIN {X 0,Y 199.39,Z 183.613,A -85,B 0,C 180,E1 -21793.438,E2 -21793.438} C_VEL
LIN {X 0,Y 201.91,Z 185.744,A -85,B 0,C 180,E1 -21795.132,E2 -21795.132} C_VEL
LIN {X 0,Y 203,Z 187.47,A -85,B 0,C 180,E1 -21795.885,E2 -21795.885} C_VEL
LIN {X 0,Y 205.338,Z 190.422,A -85,B 0,C 180,E1 -21797.347,E2 -21797.347} C_VEL
LIN {X 0,Y 206.422,Z 191.632,A -85,B 0,C 180,E1 -21797.971,E2 -21797.971} C_VEL
LIN {X 0,Y 209.181,Z 195.333,A -85,B 0,C 180,E1 -21799.519,E2 -21799.519} C_VEL
LIN {X 0,Y 210.928,Z 197.669,A -85,B 0,C 180,E1 -21800.445,E2 -21800.445} C_VEL
LIN {X 0,Y 213.955,Z 201.707,A -85,B 0,C 180,E1 -21801.961,E2 -21801.961} C_VEL
LIN {X 0,Y 218.931,Z 208.775,A -85,B 0,C 180,E1 -21804.27,E2 -21804.27} C_VEL
LIN {X 0,Y 224.368,Z 217.613,A -85,B 0,C 180,E1 -21806.563,E2 -21806.563} C_VEL
LIN {X 0,Y 229.966,Z 228.436,A -85,B 0,C 180,E1 -21808.788,E2 -21808.788} C_VEL
LIN {X 0,Y 232.557,Z 234.183,A -85,B 0,C 180,E1 -21809.785,E2 -21809.785} C_VEL
LIN {X 0,Y 229.769,Z 277.992,A -85,B 0,C 180,E1 -21811.153,E2 -21811.153} C_VEL
LIN {X 0,Y 227.875,Z 291.795,A -85,B 0,C 180,E1 -21811.871,E2 -21811.871} C_VEL
LIN {X 0,Y 225.554,Z 304.502,A -85,B 0,C 180,E1 -21812.929,E2 -21812.929} C_VEL
LIN {X 0,Y 222.312,Z 317.015,A -85,B 0,C 180,E1 -21814.321,E2 -21814.321} C_VEL
LIN {X 0,Y 218.896,Z 327.998,A -85,B 0,C 180,E1 -21815.947,E2 -21815.947} C_VEL
LIN {X 0,Y 214.977,Z 338.424,A -85,B 0,C 180,E1 -21817.937,E2 -21817.937} C_VEL
LIN {X 0,Y 211.194,Z 347.174,A -85,B 0,C 180,E1 -21820.059,E2 -21820.059} C_VEL
LIN {X 0,Y 206.886,Z 356.014,A -85,B 0,C 180,E1 -21822.796,E2 -21822.796} C_VEL
LIN {X 0,Y 203.148,Z 362.832,A -85,B 0,C 180,E1 -21825.528,E2 -21825.528} C_VEL
LIN {X 0,Y 200.182,Z 367.942,A -85,B 0,C 180,E1 -21828.16,E2 -21828.16} C_VEL
LIN {X 0,Y 196.762,Z 373.224,A -85,B 0,C 180,E1 -21831.793,E2 -21831.793} C_VEL
LIN {X 0,Y 194.645,Z 376.27,A -85,B 0,C 180,E1 -21834.711,E2 -21834.711} C_VEL
LIN {X 0,Y 193.294,Z 377.977,A -85,B 0,C 180,E1 -21836.949,E2 -21836.949} C_VEL
LIN {X 0,Y 192.201,Z 379.221,A -85,B 0,C 180,E1 -21839.208,E2 -21839.208} C_VEL
LIN {X 0,Y 191.209,Z 380.037,A -85,B 0,C 180,E1 -21841.898,E2 -21841.898} C_VEL
LIN {X 0,Y 190.262,Z 380.107,A -85,B 0,C 180,E1 -21846.026,E2 -21846.026} C_VEL
LIN {X 0,Y 190.035,Z 379.477,A -85,B 0,C 180,E1 -21848.295,E2 -21848.295} C_VEL
LIN {X 0,Y 189.916,Z 378.427,A -85,B 0,C 180,E1 -21850.546,E2 -21850.546} C_VEL
LIN {X 0,Y 190.131,Z 375.959,A -85,B 0,C 180,E1 -21853.954,E2 -21853.954} C_VEL
LIN {X 0,Y 190.663,Z 372.522,A -85,B 0,C 180,E1 -21857.223,E2 -21857.223} C_VEL
LIN {X 0,Y 191.47,Z 367.917,A -85,B 0,C 180,E1 -21860.493,E2 -21860.493} C_VEL
LIN {X 0,Y 192.598,Z 362.065,A -85,B 0,C 180,E1 -21863.715,E2 -21863.715} C_VEL
LIN {X 0,Y 194.189,Z 354.684,A -85,B 0,C 180,E1 -21866.888,E2 -21866.888} C_VEL
LIN {X 0,Y 196.227,Z 345.495,A -85,B 0,C 180,E1 -21870,E2 -21870} C_VEL
LIN {X 0,Y 198.304,Z 335.993,A -85,B 0,C 180,E1 -21872.539,E2 -21872.539} C_VEL
LIN {X 0,Y 200.381,Z 325.4,A -85,B 0,C 180,E1 -21874.779,E2 -21874.779} C_VEL
LIN {X 0,Y 202.215,Z 315.212,A -85,B 0,C 180,E1 -21876.486,E2 -21876.486} C_VEL
LIN {X 0,Y 203.891,Z 303.36,A -85,B 0,C 180,E1 -21878.05,E2 -21878.05} C_VEL
LIN {X 0,Y 205.389,Z 290.292,A -85,B 0,C 180,E1 -21879.292,E2 -21879.292} C_VEL
LIN {X 0,Y 206.462,Z 276.732,A -85,B 0,C 180,E1 -21880.15,E2 -21880.15} C_VEL
LIN {X 0,Y 209.144,Z 212.795,A -85,B 0,C 180,E1 -21882.339,E2 -21882.339} C_VEL
LIN {X 0,Y 204.262,Z 198.307,A -85,B 0,C 180,E1 -21883.581,E2 -21883.581} C_VEL
LIN {X 0,Y 195.838,Z 181.158,A -85,B 0,C 180,E1 -21885.57,E2 -21885.57} C_VEL
LIN {X 0,Y 192.991,Z 175.784,A -85,B 0,C 180,E1 -21886.27,E2 -21886.27} C_VEL
LIN {X 0,Y 192.699,Z 174.484,A -85,B 0,C 180,E1 -21886.42,E2 -21886.42} C_VEL
LIN {X 0,Y 192.62,Z 174.491,A -85,B 0,C 180,E1 -21889.171,E2 -21889.171} C_VEL
LIN {X 0,Y 192.605,Z 174.449,A -85,B 0,C 180,E1 -21894.188,E2 -21894.188} C_VEL
LIN {X 0,Y 192.591,Z 174.48,A -85,B 0,C 180,E1 -21898.863,E2 -21898.863} C_VEL
LIN {X 0,Y 192.592,Z 174.493,A -85,B 0,C 180,E1 -21903.188,E2 -21903.188} C_VEL
LIN {X 0,Y 192.539,Z 174.493,A -85,B 0,C 180,E1 -21908.355,E2 -21908.355} C_VEL
LIN {X 0,Y 192.483,Z 174.501,A -85,B 0,C 180,E1 -21913.095,E2 -21913.095} C_VEL
LIN {X 0,Y 192.482,Z 174.477,A -85,B 0,C 180,E1 -21916.908,E2 -21916.908} C_VEL
LIN {X 0,Y 192.541,Z 174.498,A -85,B 0,C 180,E1 -21921.647,E2 -21921.647} C_VEL
LIN {X 0,Y 192.594,Z 174.478,A -85,B 0,C 180,E1 -21926.815,E2 -21926.815} C_VEL
LIN {X 0,Y 192.619,Z 174.454,A -85,B 0,C 180,E1 -21931.686,E2 -21931.686} C_VEL
LIN {X 0,Y 192.657,Z 174.482,A -85,B 0,C 180,E1 -21936.344,E2 -21936.344} C_VEL
LIN {X 0,Y 192.696,Z 174.475,A -85,B 0,C 180,E1 -21941.493,E2 -21941.493} C_VEL
LIN {X 0,Y 192.773,Z 174.472,A -85,B 0,C 180,E1 -21947.366,E2 -21947.366} C_VEL
LIN {X 0,Y 193.025,Z 174.429,A -85,B 0,C 180,E1 -21951.627,E2 -21951.627} C_VEL
LIN {X 0,Y 193.231,Z 174.411,A -85,B 0,C 180,E1 -21957.917,E2 -21957.917} C_VEL
LIN {X 0,Y 193.417,Z 174.383,A -85,B 0,C 180,E1 -21960.001,E2 -21960.001} C_VEL
LIN {X 0,Y 192.939,Z 174.453,A -85,B 0,C 180,E1 -21964.179,E2 -21964.179} C_VEL
LIN {X 0,Y 193.028,Z 174.431,A -85,B 0,C 180,E1 -21968.375,E2 -21968.375} C_VEL
LIN {X 0,Y 192.786,Z 174.471,A -85,B 0,C 180,E1 -21972.636,E2 -21972.636} C_VEL
LIN {X 0,Y 192.707,Z 174.471,A -85,B 0,C 180,E1 -21976.964,E2 -21976.964} C_VEL
LIN {X 0,Y 192.585,Z 174.495,A -85,B 0,C 180,E1 -21981.404,E2 -21981.404} C_VEL
LIN {X 0,Y 192.64,Z 174.488,A -85,B 0,C 180,E1 -21984.206,E2 -21984.206} C_VEL
LIN {X 0,Y 192.606,Z 174.493,A -85,B 0,C 180,E1 -21988.866,E2 -21988.866} C_VEL
LIN {X 0,Y 192.599,Z 174.496,A -85,B 0,C 180,E1 -21993.187,E2 -21993.187} C_VEL
LIN {X 0,Y 192.546,Z 174.502,A -85,B 0,C 180,E1 -21998.355,E2 -21998.355} C_VEL
LIN {X 0,Y 192.489,Z 174.513,A -85,B 0,C 180,E1 -22003.094,E2 -22003.094} C_VEL
LIN {X 0,Y 192.49,Z 174.512,A -85,B 0,C 180,E1 -22006.906,E2 -22006.906} C_VEL
LIN {X 0,Y 192.53,Z 174.546,A -85,B 0,C 180,E1 -22010.271,E2 -22010.271} C_VEL
LIN {X 0,Y 194.156,Z 181.172,A -85,B 0,C 180,E1 -22013.629,E2 -22013.629} C_VEL
LIN {X 0,Y 201.339,Z 199.061,A -85,B 0,C 180,E1 -22015.506,E2 -22015.506} C_VEL
LIN {X 0,Y 205.174,Z 210.098,A -85,B 0,C 180,E1 -22016.498,E2 -22016.498} C_VEL
LIN {X 0,Y 206.515,Z 221.991,A -85,B 0,C 180,E1 -22017.15,E2 -22017.15} C_VEL
LIN {X 0,Y 206.583,Z 227.831,A -85,B 0,C 180,E1 -22017.388,E2 -22017.388} C_VEL
LIN {X 0,Y 205.581,Z 233.693,A -85,B 0,C 180,E1 -22017.485,E2 -22017.485} C_VEL
LIN {X 0,Y 202.493,Z 245.373,A -85,B 0,C 180,E1 -22017.537,E2 -22017.537} C_VEL
LIN {X 0,Y 201.463,Z 251.305,A -85,B 0,C 180,E1 -22017.636,E2 -22017.636} C_VEL
LIN {X 0,Y 201.332,Z 253.298,A -85,B 0,C 180,E1 -22017.698,E2 -22017.698} C_VEL
LIN {X 0,Y 199.672,Z 290.199,A -85,B 0,C 180,E1 -22019.017,E2 -22019.017} C_VEL
LIN {X 0,Y 198.383,Z 304.024,A -85,B 0,C 180,E1 -22019.9,E2 -22019.9} C_VEL
LIN {X 0,Y 196.611,Z 316.978,A -85,B 0,C 180,E1 -22021.146,E2 -22021.146} C_VEL
LIN {X 0,Y 194.778,Z 328.014,A -85,B 0,C 180,E1 -22022.609,E2 -22022.609} C_VEL
LIN {X 0,Y 192.816,Z 338.273,A -85,B 0,C 180,E1 -22024.352,E2 -22024.352} C_VEL
LIN {X 0,Y 190.76,Z 347.83,A -85,B 0,C 180,E1 -22026.38,E2 -22026.38} C_VEL
LIN {X 0,Y 188.828,Z 356.411,A -85,B 0,C 180,E1 -22028.631,E2 -22028.631} C_VEL
LIN {X 0,Y 187.404,Z 363.362,A -85,B 0,C 180,E1 -22030.843,E2 -22030.843} C_VEL
LIN {X 0,Y 185.61,Z 371.61,A -85,B 0,C 180,E1 -22034.066,E2 -22034.066} C_VEL
LIN {X 0,Y 184.444,Z 377.196,A -85,B 0,C 180,E1 -22036.784,E2 -22036.784} C_VEL
LIN {X 0,Y 183.681,Z 382.655,A -85,B 0,C 180,E1 -22040.085,E2 -22040.085} C_VEL
LIN {X 0,Y 183.288,Z 386.884,A -85,B 0,C 180,E1 -22043.394,E2 -22043.394} C_VEL
LIN {X 0,Y 183.163,Z 389.497,A -85,B 0,C 180,E1 -22046.067,E2 -22046.067} C_VEL
LIN {X 0,Y 183.345,Z 392.136,A -85,B 0,C 180,E1 -22050,E2 -22050} C_VEL
LIN {X 0,Y 183.079,Z 393.335,A -85,B 0,C 180,E1 -22053.53,E2 -22053.53} C_VEL
LIN {X 0,Y 183.208,Z 393.561,A -85,B 0,C 180,E1 -22056.608,E2 -22056.608} C_VEL
LIN {X 0,Y 183.98,Z 392.536,A -85,B 0,C 180,E1 -22061.011,E2 -22061.011} C_VEL
LIN {X 0,Y 184.741,Z 391.459,A -85,B 0,C 180,E1 -22063.194,E2 -22063.194} C_VEL
LIN {X 0,Y 185.675,Z 389.962,A -85,B 0,C 180,E1 -22065.364,E2 -22065.364} C_VEL
LIN {X 0,Y 187.768,Z 386.943,A -85,B 0,C 180,E1 -22068.551,E2 -22068.551} C_VEL
LIN {X 0,Y 190.394,Z 382.904,A -85,B 0,C 180,E1 -22071.662,E2 -22071.662} C_VEL
LIN {X 0,Y 193.679,Z 377.377,A -85,B 0,C 180,E1 -22074.881,E2 -22074.881} C_VEL
LIN {X 0,Y 197.843,Z 370.082,A -85,B 0,C 180,E1 -22078.078,E2 -22078.078} C_VEL
LIN {X 0,Y 202.268,Z 361.841,A -85,B 0,C 180,E1 -22080.831,E2 -22080.831} C_VEL
LIN {X 0,Y 206.326,Z 353.435,A -85,B 0,C 180,E1 -22083.025,E2 -22083.025} C_VEL
LIN {X 0,Y 210.591,Z 343.132,A -85,B 0,C 180,E1 -22085.147,E2 -22085.147} C_VEL
LIN {X 0,Y 214.888,Z 331.547,A -85,B 0,C 180,E1 -22086.939,E2 -22086.939} C_VEL
LIN {X 0,Y 218.401,Z 320.079,A -85,B 0,C 180,E1 -22088.276,E2 -22088.276} C_VEL
LIN {X 0,Y 221.488,Z 306.994,A -85,B 0,C 180,E1 -22089.391,E2 -22089.391} C_VEL
LIN {X 0,Y 223.732,Z 294.047,A -85,B 0,C 180,E1 -22090.143,E2 -22090.143} C_VEL
